gfCNCPoint3[19226] = {X 296.3838, Y 61.4413, Z -4.6667, A 0.000, B 0.000, C 0.000 }
gfCNCPoint3[19227] = {X 295.8066, Y 62.1158, Z -4.6667, A 0.000, B 0.000, C 0.000 }
gfCNCPoint3[19228] = {X 295.1062, Y 62.6612, Z -4.6667, A 0.000, B 0.000, C 0.000 }
gfCNCPoint3[19229] = {X 294.3109, Y 63.0556, Z -4.6667, A 0.000, B 0.000, C 0.000 }
gfCNCPoint3[19230] = {X 293.4528, Y 63.2829, Z -4.6667, A 0.000, B 0.000, C 0.000 }
gfCNCPoint3[19231] = {X 293.4528, Y 92.7108, Z -4.6667, A 0.000, B 0.000, C 0.000 }
gfCNCPoint3[19232] = {X 294.3107, Y 92.9407, Z -4.6667, A 0.000, B 0.000, C 0.000 }
gfCNCPoint3[19233] = {X 295.1055, Y 93.3369, Z -4.6667, A 0.000, B 0.000, C 0.000 }
gfCNCPoint3[19234] = {X 295.8055, Y 93.8837, Z -4.6667, A 0.000, B 0.000, C 0.000 }
gfCNCPoint3[19235] = {X 296.3823, Y 94.5590, Z -4.6667, A 0.000, B 0.000, C 0.000 }
gfCNCPoint3[19236] = {X 296.8130, Y 95.3358, Z -4.6667, A 0.000, B 0.000, C 0.000 }
gfCNCPoint3[19237] = {X 297.0801, Y 96.1828, Z -4.6667, A 0.000, B 0.000, C 0.000 }
gfCNCPoint3[19238] = {X 297.1731, Y 97.0661, Z -4.6667, A 0.000, B 0.000, C 0.000 }
gfCNCPoint3[19239] = {X 297.1731, Y 97.6950, Z -4.6667, A 0.000, B 0.000, C 0.000 }
gfCNCPoint3[19240] = {X 297.6531, Y 97.6950, Z -4.6667, A 0.000, B 0.000, C 0.000 }
gfCNCPoint3[19241] = {X 314.2152, Y 97.6950, Z -4.6667, A 0.000, B 0.000, C 0.000 }
gfCNCPoint3[19242] = {X 313.0166, Y 96.8446, Z -4.6667, A 0.000, B 0.000, C 0.000 }
gfCNCPoint3[19243] = {X 311.8818, Y 95.9106, Z -4.6667, A 0.000, B 0.000, C 0.000 }
gfCNCPoint3[19244] = {X 310.9060, Y 94.9487, Z -4.6667, A 0.000, B 0.000, C 0.000 }
gfCNCPoint3[19245] = {X 310.0416, Y 93.8855, Z -4.6667, A 0.000, B 0.000, C 0.000 }
gfCNCPoint3[19246] = {X 309.2076, Y 92.5708, Z -4.6667, A 0.000, B 0.000, C 0.000 }
gfCNCPoint3[19247] = {X 308.5438, Y 91.1625, Z -4.6667, A 0.000, B 0.000, C 0.000 }
gfCNCPoint3[19248] = {X 308.0605, Y 89.6826, Z -4.6667, A 0.000, B 0.000, C 0.000 }
gfCNCPoint3[19249] = {X 307.7070, Y 88.0127, Z -4.6667, A 0.000, B 0.000, C 0.000 }
gfCNCPoint3[19250] = {X 307.4982, Y 86.3187, Z -4.6667, A 0.000, B 0.000, C 0.000 }
gfCNCPoint3[19251] = {X 307.4354, Y 84.6131, Z -4.6667, A 0.000, B 0.000, C 0.000 }
gfCNCPoint3[19252] = {X 307.4366, Y 63.6743, Z -4.6667, A 0.000, B 0.000, C 0.000 }
gfCNCPoint3[19253] = {X 306.4282, Y 63.3060, Z -4.6667, A 0.000, B 0.000, C 0.000 }
gfCNCPoint3[19254] = {X 305.5247, Y 62.7262, Z -4.6667, A 0.000, B 0.000, C 0.000 }
gfCNCPoint3[19255] = {X 304.7699, Y 61.9628, Z -4.6667, A 0.000, B 0.000, C 0.000 }
gfCNCPoint3[19256] = {X 304.2002, Y 61.0529, Z -4.6667, A 0.000, B 0.000, C 0.000 }
gfCNCPoint3[19257] = {X 303.8433, Y 60.0404, Z -4.6667, A 0.000, B 0.000, C 0.000 }
gfCNCPoint3[19258] = {X 303.7164, Y 58.9744, Z -4.6667, A 0.000, B 0.000, C 0.000 }
gfCNCPoint3[19259] = {X 303.7162, Y 58.0000, Z -4.6667, A 0.000, B 0.000, C 0.000 }
gfCNCPoint3[19260] = {X 303.8100, Y 57.0480, Z -4.6667, A 0.000, B 0.000, C 0.000 }
gfCNCPoint3[19261] = {X 304.0877, Y 56.1325, Z -4.6667, A 0.000, B 0.000, C 0.000 }
gfCNCPoint3[19262] = {X 304.5387, Y 55.2888, Z -4.6667, A 0.000, B 0.000, C 0.000 }
gfCNCPoint3[19263] = {X 305.1455, Y 54.5493, Z -4.6667, A 0.000, B 0.000, C 0.000 }
gfCNCPoint3[19264] = {X 305.8850, Y 53.9424, Z -4.6667, A 0.000, B 0.000, C 0.000 }
gfCNCPoint3[19265] = {X 306.7287, Y 53.4915, Z -4.6667, A 0.000, B 0.000, C 0.000 }
gfCNCPoint3[19266] = {X 307.6442, Y 53.2138, Z -4.6667, A 0.000, B 0.000, C 0.000 }
gfCNCPoint3[19267] = {X 308.5962, Y 53.1200, Z -4.6667, A 0.000, B 0.000, C 0.000 }
gfCNCPoint3[19268] = {X 324.3107, Y 53.1200, Z -4.6667, A 0.000, B 0.000, C 0.000 }
gfCNCPoint3[19269] = {X 325.2627, Y 53.2138, Z -4.6667, A 0.000, B 0.000, C 0.000 }
gfCNCPoint3[19270] = {X 326.1782, Y 53.4915, Z -4.6667, A 0.000, B 0.000, C 0.000 }
gfCNCPoint3[19271] = {X 327.0219, Y 53.9424, Z -4.6667, A 0.000, B 0.000, C 0.000 }
gfCNCPoint3[19272] = {X 327.7614, Y 54.5493, Z -4.6667, A 0.000, B 0.000, C 0.000 }
gfCNCPoint3[19273] = {X 328.3683, Y 55.2888, Z -4.6667, A 0.000, B 0.000, C 0.000 }
gfCNCPoint3[19274] = {X 328.8192, Y 56.1325, Z -4.6667, A 0.000, B 0.000, C 0.000 }
gfCNCPoint3[19275] = {X 329.0969, Y 57.0480, Z -4.6667, A 0.000, B 0.000, C 0.000 }
gfCNCPoint3[19276] = {X 329.1907, Y 58.0000, Z -4.6667, A 0.000, B 0.000, C 0.000 }
gfCNCPoint3[19277] = {X 329.1907, Y 58.9341, Z -4.6667, A 0.000, B 0.000, C 0.000 }
gfCNCPoint3[19278] = {X 329.0671, Y 60.0067, Z -4.6667, A 0.000, B 0.000, C 0.000 }
gfCNCPoint3[19279] = {X 328.7125, Y 61.0265, Z -4.6667, A 0.000, B 0.000, C 0.000 }
gfCNCPoint3[19280] = {X 328.1440, Y 61.9444, Z -4.6667, A 0.000, B 0.000, C 0.000 }
gfCNCPoint3[19281] = {X 327.3888, Y 62.7161, Z -4.6667, A 0.000, B 0.000, C 0.000 }
gfCNCPoint3[19282] = {X 326.4835, Y 63.3044, Z -4.6667, A 0.000, B 0.000, C 0.000 }
gfCNCPoint3[19283] = {X 325.4716, Y 63.6810, Z -4.6667, A 0.000, B 0.000, C 0.000 }
gfCNCPoint3[19284] = {X 325.4732, Y 83.2268, Z -4.6667, A 0.000, B 0.000, C 0.000 }
gfCNCPoint3[19285] = {X 325.4867, Y 84.6073, Z -4.6667, A 0.000, B 0.000, C 0.000 }
gfCNCPoint3[19286] = {X 325.5527, Y 85.7200, Z -4.6667, A 0.000, B 0.000, C 0.000 }
gfCNCPoint3[19287] = {X 325.7426, Y 86.8184, Z -4.6667, A 0.000, B 0.000, C 0.000 }
gfCNCPoint3[19288] = {X 325.8866, Y 86.9525, Z -4.6667, A 0.000, B 0.000, C 0.000 }
gfCNCPoint3[19289] = {X 326.0549, Y 87.0546, Z -4.6667, A 0.000, B 0.000, C 0.000 }
gfCNCPoint3[19290] = {X 326.4838, Y 87.2970, Z -4.6667, A 0.000, B 0.000, C 0.000 }
gfCNCPoint3[19291] = {X 327.8570, Y 87.8652, Z -4.6667, A 0.000, B 0.000, C 0.000 }
gfCNCPoint3[19292] = {X 329.2839, Y 88.2806, Z -4.6667, A 0.000, B 0.000, C 0.000 }
gfCNCPoint3[19293] = {X 332.3217, Y 88.8890, Z -4.6667, A 0.000, B 0.000, C 0.000 }
gfCNCPoint3[19294] = {X 335.3954, Y 89.2771, Z -4.6667, A 0.000, B 0.000, C 0.000 }
gfCNCPoint3[19295] = {X 339.5150, Y 89.5958, Z -4.6667, A 0.000, B 0.000, C 0.000 }
gfCNCPoint3[19296] = {X 343.6430, Y 89.7746, Z -4.6667, A 0.000, B 0.000, C 0.000 }
gfCNCPoint3[19297] = {X 347.7747, Y 89.8134, Z -4.6667, A 0.000, B 0.000, C 0.000 }
gfCNCPoint3[19298] = {X 352.1399, Y 89.7754, Z -4.6667, A 0.000, B 0.000, C 0.000 }
gfCNCPoint3[19299] = {X 356.5008, Y 89.5805, Z -4.6667, A 0.000, B 0.000, C 0.000 }
gfCNCPoint3[19300] = {X 360.8519, Y 89.2288, Z -4.6667, A 0.000, B 0.000, C 0.000 }
gfCNCPoint3[19301] = {X 363.1336, Y 88.9451, Z -4.6667, A 0.000, B 0.000, C 0.000 }
gfCNCPoint3[19302] = {X 365.3941, Y 88.5248, Z -4.6667, A 0.000, B 0.000, C 0.000 }
gfCNCPoint3[19303] = {X 367.6252, Y 87.9694, Z -4.6667, A 0.000, B 0.000, C 0.000 }
gfCNCPoint3[19304] = {X 368.9185, Y 87.4946, Z -4.6667, A 0.000, B 0.000, C 0.000 }
gfCNCPoint3[19305] = {X 370.1140, Y 86.8097, Z -4.6667, A 0.000, B 0.000, C 0.000 }
gfCNCPoint3[19306] = {X 370.2985, Y 85.3241, Z -4.6667, A 0.000, B 0.000, C 0.000 }
gfCNCPoint3[19307] = {X 370.3601, Y 83.8283, Z -4.6667, A 0.000, B 0.000, C 0.000 }
gfCNCPoint3[19308] = {X 370.3587, Y 63.6740, Z -4.6667, A 0.000, B 0.000, C 0.000 }
gfCNCPoint3[19309] = {X 369.3505, Y 63.3056, Z -4.6667, A 0.000, B 0.000, C 0.000 }
gfCNCPoint3[19310] = {X 368.4472, Y 62.7258, Z -4.6667, A 0.000, B 0.000, C 0.000 }
gfCNCPoint3[19311] = {X 367.6926, Y 61.9624, Z -4.6667, A 0.000, B 0.000, C 0.000 }
gfCNCPoint3[19312] = {X 367.1231, Y 61.0526, Z -4.6667, A 0.000, B 0.000, C 0.000 }
gfCNCPoint3[19313] = {X 366.7663, Y 60.0402, Z -4.6667, A 0.000, B 0.000, C 0.000 }
gfCNCPoint3[19314] = {X 366.6394, Y 58.9744, Z -4.6667, A 0.000, B 0.000, C 0.000 }
gfCNCPoint3[19315] = {X 366.6393, Y 58.0000, Z -4.6667, A 0.000, B 0.000, C 0.000 }
gfCNCPoint3[19316] = {X 366.7331, Y 57.0480, Z -4.6667, A 0.000, B 0.000, C 0.000 }
gfCNCPoint3[19317] = {X 367.0108, Y 56.1325, Z -4.6667, A 0.000, B 0.000, C 0.000 }
gfCNCPoint3[19318] = {X 367.4617, Y 55.2888, Z -4.6667, A 0.000, B 0.000, C 0.000 }
gfCNCPoint3[19319] = {X 368.0686, Y 54.5493, Z -4.6667, A 0.000, B 0.000, C 0.000 }
gfCNCPoint3[19320] = {X 368.8081, Y 53.9424, Z -4.6667, A 0.000, B 0.000, C 0.000 }
gfCNCPoint3[19321] = {X 369.6518, Y 53.4915, Z -4.6667, A 0.000, B 0.000, C 0.000 }
gfCNCPoint3[19322] = {X 370.5672, Y 53.2138, Z -4.6667, A 0.000, B 0.000, C 0.000 }
gfCNCPoint3[19323] = {X 371.5193, Y 53.1200, Z -4.6667, A 0.000, B 0.000, C 0.000 }
gfCNCPoint3[19324] = {X 388.0597, Y 53.1200, Z -4.6667, A 0.000, B 0.000, C 0.000 }
gfCNCPoint3[19325] = {X 389.0355, Y 53.2186, Z -4.6667, A 0.000, B 0.000, C 0.000 }
gfCNCPoint3[19326] = {X 389.9719, Y 53.5102, Z -4.6667, A 0.000, B 0.000, C 0.000 }
gfCNCPoint3[19327] = {X 390.8310, Y 53.9833, Z -4.6667, A 0.000, B 0.000, C 0.000 }
gfCNCPoint3[19328] = {X 391.5783, Y 54.6186, Z -4.6667, A 0.000, B 0.000, C 0.000 }
gfCNCPoint3[19329] = {X 392.1572, Y 55.3496, Z -4.6667, A 0.000, B 0.000, C 0.000 }
gfCNCPoint3[19330] = {X 392.5865, Y 56.1774, Z -4.6667, A 0.000, B 0.000, C 0.000 }
gfCNCPoint3[19331] = {X 392.8506, Y 57.0718, Z -4.6667, A 0.000, B 0.000, C 0.000 }
gfCNCPoint3[19332] = {X 392.9397, Y 58.0000, Z -4.6667, A 0.000, B 0.000, C 0.000 }
gfCNCPoint3[19333] = {X 392.9395, Y 58.9743, Z -4.6667, A 0.000, B 0.000, C 0.000 }
gfCNCPoint3[19334] = {X 392.8783, Y 59.7057, Z -4.6667, A 0.000, B 0.000, C 0.000 }
gfCNCPoint3[19335] = {X 392.7080, Y 60.4197, Z -4.6667, A 0.000, B 0.000, C 0.000 }
gfCNCPoint3[19336] = {X 392.4327, Y 61.1000, Z -4.6667, A 0.000, B 0.000, C 0.000 }
gfCNCPoint3[19337] = {X 392.0515, Y 61.7416, Z -4.6667, A 0.000, B 0.000, C 0.000 }
gfCNCPoint3[19338] = {X 391.5775, Y 62.3178, Z -4.6667, A 0.000, B 0.000, C 0.000 }
gfCNCPoint3[19339] = {X 390.8819, Y 62.9185, Z -4.6667, A 0.000, B 0.000, C 0.000 }
gfCNCPoint3[19340] = {X 390.0864, Y 63.3788, Z -4.6667, A 0.000, B 0.000, C 0.000 }
gfCNCPoint3[19341] = {X 389.2190, Y 63.6825, Z -4.6667, A 0.000, B 0.000, C 0.000 }
gfCNCPoint3[19342] = {X 389.2180, Y 73.4816, Z -4.6667, A 0.000, B 0.000, C 0.000 }
gfCNCPoint3[19343] = {X 398.8180, Y 73.4825, Z -4.6667, A 0.000, B 0.000, C 0.000 }
gfCNCPoint3[19344] = {X 398.8173, Y 80.5578, Z -4.6667, A 0.000, B 0.000, C 0.000 }
gfCNCPoint3[19345] = {X 405.8037, Y 76.0835, Z -4.6667, A 0.000, B 0.000, C 0.000 }
gfCNCPoint3[19346] = {X 400.0374, Y 73.8211, Z -4.6667, A 0.000, B 0.000, C 0.000 }
gfCNCPoint3[19347] = {X 399.4365, Y 73.6201, Z -4.6667, A 0.000, B 0.000, C 0.000 }
gfCNCPoint3[19348] = {X 398.8180, Y 73.4825, Z -4.6667, A 0.000, B 0.000, C 0.000 }
gfCNCPoint3[19349] = {X 396.4180, Y 73.4822, Z -4.6667, A 0.000, B 0.000, C 0.000 }
gfCNCPoint3[19350] = {X 396.4170, Y 84.5897, Z -4.6667, A 0.000, B 0.000, C 0.000 }
gfCNCPoint3[19351] = {X 396.4168, Y 84.9452, Z -4.6667, A 0.000, B 0.000, C 0.000 }
gfCNCPoint3[19352] = {X 411.0595, Y 75.5675, Z -4.6667, A 0.000, B 0.000, C 0.000 }
gfCNCPoint3[19353] = {X 400.9158, Y 71.5876, Z -4.6667, A 0.000, B 0.000, C 0.000 }
gfCNCPoint3[19354] = {X 399.6202, Y 71.1939, Z -4.6667, A 0.000, B 0.000, C 0.000 }
gfCNCPoint3[19355] = {X 398.2786, Y 71.0108, Z -4.6667, A 0.000, B 0.000, C 0.000 }
gfCNCPoint3[19356] = {X 397.3448, Y 70.9530, Z -4.6667, A 0.000, B 0.000, C 0.000 }
gfCNCPoint3[19357] = {X 396.4183, Y 70.8231, Z -4.6667, A 0.000, B 0.000, C 0.000 }
gfCNCPoint3[19358] = {X 396.4180, Y 73.4822, Z -4.6667, A 0.000, B 0.000, C 0.000 }
gfCNCPoint3[19359] = {X 394.0180, Y 73.4820, Z -4.6667, A 0.000, B 0.000, C 0.000 }
gfCNCPoint3[19360] = {X 394.0170, Y 84.5974, Z -4.6667, A 0.000, B 0.000, C 0.000 }
gfCNCPoint3[19361] = {X 394.0175, Y 84.7629, Z -4.6667, A 0.000, B 0.000, C 0.000 }
gfCNCPoint3[19362] = {X 394.0169, Y 84.9284, Z -4.6667, A 0.000, B 0.000, C 0.000 }
gfCNCPoint3[19363] = {X 393.9665, Y 86.3336, Z -4.6667, A 0.000, B 0.000, C 0.000 }
gfCNCPoint3[19364] = {X 393.8352, Y 87.7335, Z -4.6667, A 0.000, B 0.000, C 0.000 }
gfCNCPoint3[19365] = {X 395.0900, Y 87.4758, Z -4.6667, A 0.000, B 0.000, C 0.000 }
gfCNCPoint3[19366] = {X 396.3680, Y 87.3860, Z -4.6667, A 0.000, B 0.000, C 0.000 }
gfCNCPoint3[19367] = {X 396.7432, Y 87.3712, Z -4.6667, A 0.000, B 0.000, C 0.000 }
gfCNCPoint3[19368] = {X 397.1178, Y 87.3462, Z -4.6667, A 0.000, B 0.000, C 0.000 }
gfCNCPoint3[19369] = {X 416.3153, Y 75.0514, Z -4.6667, A 0.000, B 0.000, C 0.000 }
gfCNCPoint3[19370] = {X 401.7941, Y 69.3541, Z -4.6667, A 0.000, B 0.000, C 0.000 }
gfCNCPoint3[19371] = {X 400.6812, Y 68.9842, Z -4.6667, A 0.000, B 0.000, C 0.000 }
gfCNCPoint3[19372] = {X 399.5351, Y 68.7359, Z -4.6667, A 0.000, B 0.000, C 0.000 }
gfCNCPoint3[19373] = {X 398.3689, Y 68.6122, Z -4.6667, A 0.000, B 0.000, C 0.000 }
gfCNCPoint3[19374] = {X 397.6031, Y 68.5669, Z -4.6667, A 0.000, B 0.000, C 0.000 }
gfCNCPoint3[19375] = {X 396.8433, Y 68.4610, Z -4.6667, A 0.000, B 0.000, C 0.000 }
gfCNCPoint3[19376] = {X 395.3930, Y 68.0821, Z -4.6667, A 0.000, B 0.000, C 0.000 }
gfCNCPoint3[19377] = {X 394.0186, Y 67.4838, Z -4.6667, A 0.000, B 0.000, C 0.000 }
gfCNCPoint3[19378] = {X 394.0180, Y 73.4820, Z -4.6667, A 0.000, B 0.000, C 0.000 }
gfCNCPoint3[19379] = {X 391.6180, Y 73.4818, Z -4.6667, A 0.000, B 0.000, C 0.000 }
gfCNCPoint3[19380] = {X 391.6169, Y 84.6054, Z -4.6667, A 0.000, B 0.000, C 0.000 }
gfCNCPoint3[19381] = {X 391.5809, Y 86.0256, Z -4.6667, A 0.000, B 0.000, C 0.000 }
gfCNCPoint3[19382] = {X 391.4531, Y 87.4405, Z -4.6667, A 0.000, B 0.000, C 0.000 }
gfCNCPoint3[19383] = {X 391.2288, Y 88.8722, Z -4.6667, A 0.000, B 0.000, C 0.000 }
gfCNCPoint3[19384] = {X 390.9106, Y 90.2860, Z -4.6667, A 0.000, B 0.000, C 0.000 }
gfCNCPoint3[19385] = {X 390.3344, Y 92.0499, Z -4.6667, A 0.000, B 0.000, C 0.000 }
gfCNCPoint3[19386] = {X 389.5429, Y 93.7283, Z -4.6667, A 0.000, B 0.000, C 0.000 }
gfCNCPoint3[19387] = {X 388.5486, Y 95.2950, Z -4.6667, A 0.000, B 0.000, C 0.000 }
gfCNCPoint3[19388] = {X 389.3446, Y 95.2950, Z -4.6667, A 0.000, B 0.000, C 0.000 }
gfCNCPoint3[19389] = {X 389.7639, Y 94.0857, Z -4.6667, A 0.000, B 0.000, C 0.000 }
gfCNCPoint3[19390] = {X 390.3885, Y 92.9685, Z -4.6667, A 0.000, B 0.000, C 0.000 }
gfCNCPoint3[19391] = {X 391.1991, Y 91.9779, Z -4.6667, A 0.000, B 0.000, C 0.000 }
gfCNCPoint3[19392] = {X 392.1707, Y 91.1447, Z -4.6667, A 0.000, B 0.000, C 0.000 }
gfCNCPoint3[19393] = {X 393.2732, Y 90.4945, Z -4.6667, A 0.000, B 0.000, C 0.000 }
gfCNCPoint3[19394] = {X 394.4725, Y 90.0474, Z -4.6667, A 0.000, B 0.000, C 0.000 }
gfCNCPoint3[19395] = {X 395.4279, Y 89.8519, Z -4.6667, A 0.000, B 0.000, C 0.000 }
gfCNCPoint3[19396] = {X 396.4007, Y 89.7859, Z -4.6667, A 0.000, B 0.000, C 0.000 }
gfCNCPoint3[19397] = {X 397.1636, Y 89.7496, Z -4.6667, A 0.000, B 0.000, C 0.000 }
gfCNCPoint3[19398] = {X 397.9239, Y 89.6774, Z -4.6667, A 0.000, B 0.000, C 0.000 }
gfCNCPoint3[19399] = {X 417.6096, Y 77.0725, Z -4.6667, A 0.000, B 0.000, C 0.000 }
gfCNCPoint3[19400] = {X 421.5711, Y 74.5354, Z -4.6667, A 0.000, B 0.000, C 0.000 }
gfCNCPoint3[19401] = {X 402.6725, Y 67.1206, Z -4.6667, A 0.000, B 0.000, C 0.000 }
gfCNCPoint3[19402] = {X 401.3007, Y 66.6655, Z -4.6667, A 0.000, B 0.000, C 0.000 }
gfCNCPoint3[19403] = {X 399.8876, Y 66.3618, Z -4.6667, A 0.000, B 0.000, C 0.000 }
gfCNCPoint3[19404] = {X 398.4499, Y 66.2133, Z -4.6667, A 0.000, B 0.000, C 0.000 }
gfCNCPoint3[19405] = {X 397.3054, Y 66.1055, Z -4.6667, A 0.000, B 0.000, C 0.000 }
gfCNCPoint3[19406] = {X 396.1922, Y 65.8190, Z -4.6667, A 0.000, B 0.000, C 0.000 }
gfCNCPoint3[19407] = {X 395.1380, Y 65.3609, Z -4.6667, A 0.000, B 0.000, C 0.000 }
gfCNCPoint3[19408] = {X 394.1690, Y 64.7424, Z -4.6667, A 0.000, B 0.000, C 0.000 }
gfCNCPoint3[19409] = {X 393.3094, Y 63.9792, Z -4.6667, A 0.000, B 0.000, C 0.000 }
gfCNCPoint3[19410] = {X 392.5123, Y 64.6964, Z -4.6667, A 0.000, B 0.000, C 0.000 }
gfCNCPoint3[19411] = {X 391.6188, Y 65.2892, Z -4.6667, A 0.000, B 0.000, C 0.000 }
gfCNCPoint3[19412] = {X 391.6180, Y 73.4818, Z -4.6667, A 0.000, B 0.000, C 0.000 }
gfCNCPoint3[19413] = {X 389.2180, Y 73.4816, Z -4.6667, A 0.000, B 0.000, C 0.000 }
gfCNCPoint3[19414] = {X 389.2169, Y 84.6139, Z -4.6667, A 0.000, B 0.000, C 0.000 }
gfCNCPoint3[19415] = {X 389.1551, Y 86.3199, Z -4.6667, A 0.000, B 0.000, C 0.000 }
gfCNCPoint3[19416] = {X 388.9447, Y 88.0140, Z -4.6667, A 0.000, B 0.000, C 0.000 }
gfCNCPoint3[19417] = {X 388.5875, Y 89.6833, Z -4.6667, A 0.000, B 0.000, C 0.000 }
gfCNCPoint3[19418] = {X 388.1043, Y 91.1629, Z -4.6667, A 0.000, B 0.000, C 0.000 }
gfCNCPoint3[19419] = {X 387.4405, Y 92.5708, Z -4.6667, A 0.000, B 0.000, C 0.000 }
gfCNCPoint3[19420] = {X 386.6065, Y 93.8850, Z -4.6667, A 0.000, B 0.000, C 0.000 }
gfCNCPoint3[19421] = {X 385.8743, Y 94.7997, Z -4.6667, A 0.000, B 0.000, C 0.000 }
gfCNCPoint3[19422] = {X 385.0595, Y 95.6417, Z -4.6667, A 0.000, B 0.000, C 0.000 }
gfCNCPoint3[19423] = {X 383.7996, Y 96.7249, Z -4.6667, A 0.000, B 0.000, C 0.000 }
gfCNCPoint3[19424] = {X 382.4506, Y 97.6950, Z -4.6667, A 0.000, B 0.000, C 0.000 }
gfCNCPoint3[19425] = {X 382.1875, Y 97.2936, Z -4.6667, A 0.000, B 0.000, C 0.000 }
gfCNCPoint3[19426] = {X 381.0199, Y 97.9993, Z -4.6667, A 0.000, B 0.000, C 0.000 }
gfCNCPoint3[19427] = {X 379.8040, Y 98.6181, Z -4.6667, A 0.000, B 0.000, C 0.000 }
gfCNCPoint3[19428] = {X 377.5271, Y 99.5766, Z -4.6667, A 0.000, B 0.000, C 0.000 }
gfCNCPoint3[19429] = {X 375.1871, Y 100.3689, Z -4.6667, A 0.000, B 0.000, C 0.000 }
gfCNCPoint3[19430] = {X 372.7962, Y 100.9907, Z -4.6667, A 0.000, B 0.000, C 0.000 }
gfCNCPoint3[19431] = {X 368.8820, Y 101.7454, Z -4.6667, A 0.000, B 0.000, C 0.000 }
gfCNCPoint3[19432] = {X 364.9353, Y 102.3062, Z -4.6667, A 0.000, B 0.000, C 0.000 }
gfCNCPoint3[19433] = {X 360.9658, Y 102.6716, Z -4.6667, A 0.000, B 0.000, C 0.000 }
gfCNCPoint3[19434] = {X 355.2455, Y 102.9767, Z -4.6667, A 0.000, B 0.000, C 0.000 }
gfCNCPoint3[19435] = {X 349.5185, Y 103.1068, Z -4.6667, A 0.000, B 0.000, C 0.000 }
gfCNCPoint3[19436] = {X 343.7903, Y 103.0618, Z -4.6667, A 0.000, B 0.000, C 0.000 }
gfCNCPoint3[19437] = {X 338.0661, Y 102.8417, Z -4.6667, A 0.000, B 0.000, C 0.000 }
gfCNCPoint3[19438] = {X 334.1085, Y 102.5645, Z -4.6667, A 0.000, B 0.000, C 0.000 }
gfCNCPoint3[19439] = {X 330.1660, Y 102.1223, Z -4.6667, A 0.000, B 0.000, C 0.000 }
gfCNCPoint3[19440] = {X 326.2454, Y 101.5158, Z -4.6667, A 0.000, B 0.000, C 0.000 }
gfCNCPoint3[19441] = {X 323.3898, Y 100.9107, Z -4.6667, A 0.000, B 0.000, C 0.000 }
gfCNCPoint3[19442] = {X 320.5867, Y 100.0961, Z -4.6667, A 0.000, B 0.000, C 0.000 }
gfCNCPoint3[19443] = {X 317.8516, Y 99.0765, Z -4.6667, A 0.000, B 0.000, C 0.000 }
gfCNCPoint3[19444] = {X 316.3332, Y 98.3751, Z -4.6667, A 0.000, B 0.000, C 0.000 }
gfCNCPoint3[19445] = {X 314.8785, Y 97.5498, Z -4.6667, A 0.000, B 0.000, C 0.000 }
gfCNCPoint3[19446] = {X 313.4975, Y 96.6063, Z -4.6667, A 0.000, B 0.000, C 0.000 }
gfCNCPoint3[19447] = {X 312.1998, Y 95.5512, Z -4.6667, A 0.000, B 0.000, C 0.000 }
gfCNCPoint3[19448] = {X 311.1892, Y 94.5459, Z -4.6667, A 0.000, B 0.000, C 0.000 }
gfCNCPoint3[19449] = {X 310.3050, Y 93.4278, Z -4.6667, A 0.000, B 0.000, C 0.000 }
gfCNCPoint3[19450] = {X 309.5595, Y 92.2128, Z -4.6667, A 0.000, B 0.000, C 0.000 }
gfCNCPoint3[19451] = {X 308.9634, Y 90.9180, Z -4.6667, A 0.000, B 0.000, C 0.000 }
gfCNCPoint3[19452] = {X 308.5250, Y 89.5616, Z -4.6667, A 0.000, B 0.000, C 0.000 }
gfCNCPoint3[19453] = {X 308.1802, Y 87.9321, Z -4.6667, A 0.000, B 0.000, C 0.000 }
gfCNCPoint3[19454] = {X 307.9765, Y 86.2791, Z -4.6667, A 0.000, B 0.000, C 0.000 }
gfCNCPoint3[19455] = {X 307.9154, Y 84.6146, Z -4.6667, A 0.000, B 0.000, C 0.000 }
gfCNCPoint3[19456] = {X 307.9166, Y 63.2813, Z -4.6667, A 0.000, B 0.000, C 0.000 }
gfCNCPoint3[19457] = {X 307.0573, Y 63.0561, Z -4.6667, A 0.000, B 0.000, C 0.000 }
gfCNCPoint3[19458] = {X 306.2606, Y 62.6630, Z -4.6667, A 0.000, B 0.000, C 0.000 }
gfCNCPoint3[19459] = {X 305.5592, Y 62.1178, Z -4.6667, A 0.000, B 0.000, C 0.000 }
gfCNCPoint3[19460] = {X 304.9816, Y 61.4429, Z -4.6667, A 0.000, B 0.000, C 0.000 }
gfCNCPoint3[19461] = {X 304.5513, Y 60.6657, Z -4.6667, A 0.000, B 0.000, C 0.000 }
gfCNCPoint3[19462] = {X 304.2859, Y 59.8179, Z -4.6667, A 0.000, B 0.000, C 0.000 }
gfCNCPoint3[19463] = {X 304.1962, Y 58.9341, Z -4.6667, A 0.000, B 0.000, C 0.000 }
gfCNCPoint3[19464] = {X 304.1962, Y 58.0000, Z -4.6667, A 0.000, B 0.000, C 0.000 }
gfCNCPoint3[19465] = {X 304.3065, Y 57.0209, Z -4.6667, A 0.000, B 0.000, C 0.000 }
gfCNCPoint3[19466] = {X 304.6320, Y 56.0909, Z -4.6667, A 0.000, B 0.000, C 0.000 }
gfCNCPoint3[19467] = {X 305.1562, Y 55.2566, Z -4.6667, A 0.000, B 0.000, C 0.000 }
gfCNCPoint3[19468] = {X 305.8529, Y 54.5599, Z -4.6667, A 0.000, B 0.000, C 0.000 }
gfCNCPoint3[19469] = {X 306.6871, Y 54.0357, Z -4.6667, A 0.000, B 0.000, C 0.000 }
gfCNCPoint3[19470] = {X 307.6171, Y 53.7103, Z -4.6667, A 0.000, B 0.000, C 0.000 }
gfCNCPoint3[19471] = {X 308.5962, Y 53.6000, Z -4.6667, A 0.000, B 0.000, C 0.000 }
gfCNCPoint3[19472] = {X 324.3107, Y 53.6000, Z -4.6667, A 0.000, B 0.000, C 0.000 }
gfCNCPoint3[19473] = {X 325.2898, Y 53.7103, Z -4.6667, A 0.000, B 0.000, C 0.000 }
gfCNCPoint3[19474] = {X 326.2198, Y 54.0357, Z -4.6667, A 0.000, B 0.000, C 0.000 }
gfCNCPoint3[19475] = {X 327.0540, Y 54.5599, Z -4.6667, A 0.000, B 0.000, C 0.000 }
gfCNCPoint3[19476] = {X 327.7507, Y 55.2566, Z -4.6667, A 0.000, B 0.000, C 0.000 }
gfCNCPoint3[19477] = {X 328.2750, Y 56.0909, Z -4.6667, A 0.000, B 0.000, C 0.000 }
gfCNCPoint3[19478] = {X 328.6004, Y 57.0209, Z -4.6667, A 0.000, B 0.000, C 0.000 }
gfCNCPoint3[19479] = {X 328.7107, Y 58.0000, Z -4.6667, A 0.000, B 0.000, C 0.000 }
gfCNCPoint3[19480] = {X 328.7107, Y 58.9364, Z -4.6667, A 0.000, B 0.000, C 0.000 }
gfCNCPoint3[19481] = {X 328.6169, Y 59.8191, Z -4.6667, A 0.000, B 0.000, C 0.000 }
gfCNCPoint3[19482] = {X 328.3493, Y 60.6655, Z -4.6667, A 0.000, B 0.000, C 0.000 }
gfCNCPoint3[19483] = {X 327.9186, Y 61.4417, Z -4.6667, A 0.000, B 0.000, C 0.000 }
gfCNCPoint3[19484] = {X 327.3421, Y 62.1166, Z -4.6667, A 0.000, B 0.000, C 0.000 }
gfCNCPoint3[19485] = {X 326.6428, Y 62.6634, Z -4.6667, A 0.000, B 0.000, C 0.000 }
gfCNCPoint3[19486] = {X 325.8487, Y 63.0601, Z -4.6667, A 0.000, B 0.000, C 0.000 }
gfCNCPoint3[19487] = {X 324.9916, Y 63.2908, Z -4.6667, A 0.000, B 0.000, C 0.000 }
gfCNCPoint3[19488] = {X 324.9932, Y 83.2292, Z -4.6667, A 0.000, B 0.000, C 0.000 }
gfCNCPoint3[19489] = {X 325.0068, Y 84.6144, Z -4.6667, A 0.000, B 0.000, C 0.000 }
gfCNCPoint3[19490] = {X 325.0826, Y 85.8324, Z -4.6667, A 0.000, B 0.000, C 0.000 }
gfCNCPoint3[19491] = {X 325.3002, Y 87.0333, Z -4.6667, A 0.000, B 0.000, C 0.000 }
gfCNCPoint3[19492] = {X 325.5332, Y 87.2838, Z -4.6667, A 0.000, B 0.000, C 0.000 }
gfCNCPoint3[19493] = {X 325.8187, Y 87.4724, Z -4.6667, A 0.000, B 0.000, C 0.000 }
gfCNCPoint3[19494] = {X 326.2616, Y 87.7228, Z -4.6667, A 0.000, B 0.000, C 0.000 }
gfCNCPoint3[19495] = {X 327.6911, Y 88.3157, Z -4.6667, A 0.000, B 0.000, C 0.000 }
gfCNCPoint3[19496] = {X 329.1769, Y 88.7485, Z -4.6667, A 0.000, B 0.000, C 0.000 }
gfCNCPoint3[19497] = {X 332.2475, Y 89.3632, Z -4.6667, A 0.000, B 0.000, C 0.000 }
gfCNCPoint3[19498] = {X 335.3543, Y 89.7554, Z -4.6667, A 0.000, B 0.000, C 0.000 }
gfCNCPoint3[19499] = {X 339.4910, Y 90.0752, Z -4.6667, A 0.000, B 0.000, C 0.000 }
gfCNCPoint3[19500] = {X 343.6362, Y 90.2546, Z -4.6667, A 0.000, B 0.000, C 0.000 }
gfCNCPoint3[19501] = {X 347.7851, Y 90.2934, Z -4.6667, A 0.000, B 0.000, C 0.000 }
gfCNCPoint3[19502] = {X 352.1632, Y 90.2549, Z -4.6667, A 0.000, B 0.000, C 0.000 }
gfCNCPoint3[19503] = {X 356.5371, Y 90.0591, Z -4.6667, A 0.000, B 0.000, C 0.000 }
gfCNCPoint3[19504] = {X 360.9012, Y 89.7062, Z -4.6667, A 0.000, B 0.000, C 0.000 }
gfCNCPoint3[19505] = {X 363.2108, Y 89.4189, Z -4.6667, A 0.000, B 0.000, C 0.000 }
gfCNCPoint3[19506] = {X 365.4989, Y 88.9933, Z -4.6667, A 0.000, B 0.000, C 0.000 }
gfCNCPoint3[19507] = {X 367.7574, Y 88.4308, Z -4.6667, A 0.000, B 0.000, C 0.000 }
gfCNCPoint3[19508] = {X 368.6801, Y 88.1205, Z -4.6667, A 0.000, B 0.000, C 0.000 }
gfCNCPoint3[19509] = {X 369.5623, Y 87.7087, Z -4.6667, A 0.000, B 0.000, C 0.000 }
gfCNCPoint3[19510] = {X 370.3927, Y 87.2006, Z -4.6667, A 0.000, B 0.000, C 0.000 }
gfCNCPoint3[19511] = {X 370.5205, Y 87.0676, Z -4.6667, A 0.000, B 0.000, C 0.000 }
gfCNCPoint3[19512] = {X 370.5863, Y 86.8954, Z -4.6667, A 0.000, B 0.000, C 0.000 }
gfCNCPoint3[19513] = {X 370.7766, Y 85.3671, Z -4.6667, A 0.000, B 0.000, C 0.000 }
gfCNCPoint3[19514] = {X 370.8401, Y 83.8283, Z -4.6667, A 0.000, B 0.000, C 0.000 }
gfCNCPoint3[19515] = {X 370.8386, Y 63.2811, Z -4.6667, A 0.000, B 0.000, C 0.000 }
gfCNCPoint3[19516] = {X 369.9795, Y 63.0558, Z -4.6667, A 0.000, B 0.000, C 0.000 }
gfCNCPoint3[19517] = {X 369.1830, Y 62.6626, Z -4.6667, A 0.000, B 0.000, C 0.000 }
gfCNCPoint3[19518] = {X 368.4818, Y 62.1174, Z -4.6667, A 0.000, B 0.000, C 0.000 }
gfCNCPoint3[19519] = {X 367.9044, Y 61.4425, Z -4.6667, A 0.000, B 0.000, C 0.000 }
gfCNCPoint3[19520] = {X 367.4742, Y 60.6654, Z -4.6667, A 0.000, B 0.000, C 0.000 }
gfCNCPoint3[19521] = {X 367.2089, Y 59.8177, Z -4.6667, A 0.000, B 0.000, C 0.000 }
gfCNCPoint3[19522] = {X 367.1193, Y 58.9340, Z -4.6667, A 0.000, B 0.000, C 0.000 }
gfCNCPoint3[19523] = {X 367.1193, Y 58.0000, Z -4.6667, A 0.000, B 0.000, C 0.000 }
gfCNCPoint3[19524] = {X 367.2296, Y 57.0209, Z -4.6667, A 0.000, B 0.000, C 0.000 }
gfCNCPoint3[19525] = {X 367.5550, Y 56.0909, Z -4.6667, A 0.000, B 0.000, C 0.000 }
gfCNCPoint3[19526] = {X 368.0792, Y 55.2566, Z -4.6667, A 0.000, B 0.000, C 0.000 }
gfCNCPoint3[19527] = {X 368.7759, Y 54.5599, Z -4.6667, A 0.000, B 0.000, C 0.000 }
gfCNCPoint3[19528] = {X 369.6102, Y 54.0357, Z -4.6667, A 0.000, B 0.000, C 0.000 }
gfCNCPoint3[19529] = {X 370.5402, Y 53.7103, Z -4.6667, A 0.000, B 0.000, C 0.000 }
gfCNCPoint3[19530] = {X 371.5193, Y 53.6000, Z -4.6667, A 0.000, B 0.000, C 0.000 }
gfCNCPoint3[19531] = {X 388.0597, Y 53.6000, Z -4.6667, A 0.000, B 0.000, C 0.000 }
gfCNCPoint3[19532] = {X 389.0388, Y 53.7103, Z -4.6667, A 0.000, B 0.000, C 0.000 }
gfCNCPoint3[19533] = {X 389.9688, Y 54.0357, Z -4.6667, A 0.000, B 0.000, C 0.000 }
gfCNCPoint3[19534] = {X 390.8030, Y 54.5599, Z -4.6667, A 0.000, B 0.000, C 0.000 }
gfCNCPoint3[19535] = {X 391.4997, Y 55.2566, Z -4.6667, A 0.000, B 0.000, C 0.000 }
gfCNCPoint3[19536] = {X 392.0239, Y 56.0909, Z -4.6667, A 0.000, B 0.000, C 0.000 }
gfCNCPoint3[19537] = {X 392.3494, Y 57.0209, Z -4.6667, A 0.000, B 0.000, C 0.000 }
gfCNCPoint3[19538] = {X 392.4597, Y 58.0000, Z -4.6667, A 0.000, B 0.000, C 0.000 }
gfCNCPoint3[19539] = {X 392.4595, Y 58.9704, Z -4.6667, A 0.000, B 0.000, C 0.000 }
gfCNCPoint3[19540] = {X 392.3397, Y 59.9546, Z -4.6667, A 0.000, B 0.000, C 0.000 }
gfCNCPoint3[19541] = {X 392.0025, Y 60.8870, Z -4.6667, A 0.000, B 0.000, C 0.000 }
gfCNCPoint3[19542] = {X 391.5594, Y 61.6016, Z -4.6667, A 0.000, B 0.000, C 0.000 }
gfCNCPoint3[19543] = {X 390.9890, Y 62.2194, Z -4.6667, A 0.000, B 0.000, C 0.000 }
gfCNCPoint3[19544] = {X 390.3120, Y 62.7180, Z -4.6667, A 0.000, B 0.000, C 0.000 }
gfCNCPoint3[19545] = {X 389.5528, Y 63.0795, Z -4.6667, A 0.000, B 0.000, C 0.000 }
gfCNCPoint3[19546] = {X 388.7390, Y 63.2908, Z -4.6667, A 0.000, B 0.000, C 0.000 }
gfCNCPoint3[19547] = {X 388.7390, Y 83.9247, Z -4.6667, A 0.000, B 0.000, C 0.000 }
gfCNCPoint3[19548] = {X 388.7369, Y 84.6150, Z -4.6667, A 0.000, B 0.000, C 0.000 }
gfCNCPoint3[19549] = {X 388.6767, Y 86.2799, Z -4.6667, A 0.000, B 0.000, C 0.000 }
gfCNCPoint3[19550] = {X 388.4716, Y 87.9333, Z -4.6667, A 0.000, B 0.000, C 0.000 }
gfCNCPoint3[19551] = {X 388.1230, Y 89.5625, Z -4.6667, A 0.000, B 0.000, C 0.000 }
gfCNCPoint3[19552] = {X 387.5872, Y 91.1606, Z -4.6667, A 0.000, B 0.000, C 0.000 }
gfCNCPoint3[19553] = {X 386.8325, Y 92.6678, Z -4.6667, A 0.000, B 0.000, C 0.000 }
gfCNCPoint3[19554] = {X 385.8739, Y 94.0542, Z -4.6667, A 0.000, B 0.000, C 0.000 }
gfCNCPoint3[19555] = {X 384.7302, Y 95.2924, Z -4.6667, A 0.000, B 0.000, C 0.000 }
gfCNCPoint3[19556] = {X 383.5022, Y 96.3481, Z -4.6667, A 0.000, B 0.000, C 0.000 }
gfCNCPoint3[19557] = {X 382.1875, Y 97.2936, Z -4.6667, A 0.000, B 0.000, C 0.000 }
gfCNCPoint3[19558] = {X 382.4506, Y 97.6950, Z -4.6667, A 0.000, B 0.000, C 0.000 }
gfCNCPoint3[19559] = {X 391.5259, Y 97.6950, Z -4.6667, A 0.000, B 0.000, C 0.000 }
gfCNCPoint3[19560] = {X 391.5259, Y 97.0659, Z -4.6667, A 0.000, B 0.000, C 0.000 }
gfCNCPoint3[19561] = {X 391.6202, Y 96.1114, Z -4.6667, A 0.000, B 0.000, C 0.000 }
gfCNCPoint3[19562] = {X 391.8994, Y 95.1937, Z -4.6667, A 0.000, B 0.000, C 0.000 }
gfCNCPoint3[19563] = {X 392.3527, Y 94.3483, Z -4.6667, A 0.000, B 0.000, C 0.000 }
gfCNCPoint3[19564] = {X 392.9626, Y 93.6079, Z -4.6667, A 0.000, B 0.000, C 0.000 }
gfCNCPoint3[19565] = {X 393.7055, Y 93.0012, Z -4.6667, A 0.000, B 0.000, C 0.000 }
gfCNCPoint3[19566] = {X 394.5528, Y 92.5515, Z -4.6667, A 0.000, B 0.000, C 0.000 }
gfCNCPoint3[19567] = {X 395.4717, Y 92.2762, Z -4.6667, A 0.000, B 0.000, C 0.000 }
gfCNCPoint3[19568] = {X 396.4267, Y 92.1860, Z -4.6667, A 0.000, B 0.000, C 0.000 }
gfCNCPoint3[19569] = {X 397.3274, Y 92.1440, Z -4.6667, A 0.000, B 0.000, C 0.000 }
gfCNCPoint3[19570] = {X 398.2250, Y 92.0585, Z -4.6667, A 0.000, B 0.000, C 0.000 }
gfCNCPoint3[19571] = {X 398.7531, Y 91.9301, Z -4.6667, A 0.000, B 0.000, C 0.000 }
gfCNCPoint3[19572] = {X 399.2394, Y 91.6875, Z -4.6667, A 0.000, B 0.000, C 0.000 }
gfCNCPoint3[19573] = {X 426.8269, Y 74.0194, Z -4.6667, A 0.000, B 0.000, C 0.000 }
gfCNCPoint3[19574] = {X 403.5509, Y 64.8871, Z -4.6667, A 0.000, B 0.000, C 0.000 }
gfCNCPoint3[19575] = {X 401.9167, Y 64.3458, Z -4.6667, A 0.000, B 0.000, C 0.000 }
gfCNCPoint3[19576] = {X 400.2331, Y 63.9867, Z -4.6667, A 0.000, B 0.000, C 0.000 }
gfCNCPoint3[19577] = {X 398.5203, Y 63.8139, Z -4.6667, A 0.000, B 0.000, C 0.000 }
gfCNCPoint3[19578] = {X 397.5546, Y 63.7099, Z -4.6667, A 0.000, B 0.000, C 0.000 }
gfCNCPoint3[19579] = {X 396.6286, Y 63.4166, Z -4.6667, A 0.000, B 0.000, C 0.000 }
gfCNCPoint3[19580] = {X 395.7791, Y 62.9457, Z -4.6667, A 0.000, B 0.000, C 0.000 }
gfCNCPoint3[19581] = {X 395.0396, Y 62.3160, Z -4.6667, A 0.000, B 0.000, C 0.000 }
gfCNCPoint3[19582] = {X 394.4660, Y 61.5934, Z -4.6667, A 0.000, B 0.000, C 0.000 }
gfCNCPoint3[19583] = {X 394.0386, Y 60.7757, Z -4.6667, A 0.000, B 0.000, C 0.000 }
gfCNCPoint3[19584] = {X 393.7727, Y 59.8921, Z -4.6667, A 0.000, B 0.000, C 0.000 }
gfCNCPoint3[19585] = {X 393.6779, Y 58.9744, Z -4.6667, A 0.000, B 0.000, C 0.000 }
gfCNCPoint3[19586] = {X 393.6777, Y 58.0000, Z -4.6667, A 0.000, B 0.000, C 0.000 }
gfCNCPoint3[19587] = {X 393.7668, Y 57.0718, Z -4.6667, A 0.000, B 0.000, C 0.000 }
gfCNCPoint3[19588] = {X 394.0309, Y 56.1774, Z -4.6667, A 0.000, B 0.000, C 0.000 }
gfCNCPoint3[19589] = {X 394.4602, Y 55.3496, Z -4.6667, A 0.000, B 0.000, C 0.000 }
gfCNCPoint3[19590] = {X 395.0391, Y 54.6186, Z -4.6667, A 0.000, B 0.000, C 0.000 }
gfCNCPoint3[19591] = {X 395.7864, Y 53.9833, Z -4.6667, A 0.000, B 0.000, C 0.000 }
gfCNCPoint3[19592] = {X 396.6455, Y 53.5102, Z -4.6667, A 0.000, B 0.000, C 0.000 }
gfCNCPoint3[19593] = {X 397.5819, Y 53.2186, Z -4.6667, A 0.000, B 0.000, C 0.000 }
gfCNCPoint3[19594] = {X 398.5577, Y 53.1200, Z -4.6667, A 0.000, B 0.000, C 0.000 }
gfCNCPoint3[19595] = {X 419.4886, Y 53.1200, Z -4.6667, A 0.000, B 0.000, C 0.000 }
gfCNCPoint3[19596] = {X 420.5534, Y 53.2376, Z -4.6667, A 0.000, B 0.000, C 0.000 }
gfCNCPoint3[19597] = {X 421.5668, Y 53.5847, Z -4.6667, A 0.000, B 0.000, C 0.000 }
gfCNCPoint3[19598] = {X 422.4802, Y 54.1445, Z -4.6667, A 0.000, B 0.000, C 0.000 }
gfCNCPoint3[19599] = {X 423.2493, Y 54.8901, Z -4.6667, A 0.000, B 0.000, C 0.000 }
gfCNCPoint3[19600] = {X 423.8373, Y 55.7856, Z -4.6667, A 0.000, B 0.000, C 0.000 }
gfCNCPoint3[19601] = {X 424.2157, Y 56.7878, Z -4.6667, A 0.000, B 0.000, C 0.000 }
gfCNCPoint3[19602] = {X 424.3662, Y 57.8484, Z -4.6667, A 0.000, B 0.000, C 0.000 }
gfCNCPoint3[19603] = {X 429.8190, Y 59.9732, Z -4.6667, A 0.000, B 0.000, C 0.000 }
gfCNCPoint3[19604] = {X 457.2986, Y 70.8760, Z -4.6667, A 0.000, B 0.000, C 0.000 }
gfCNCPoint3[19605] = {X 457.2990, Y 63.6740, Z -4.6667, A 0.000, B 0.000, C 0.000 }
gfCNCPoint3[19606] = {X 456.2908, Y 63.3057, Z -4.6667, A 0.000, B 0.000, C 0.000 }
gfCNCPoint3[19607] = {X 455.3876, Y 62.7258, Z -4.6667, A 0.000, B 0.000, C 0.000 }
gfCNCPoint3[19608] = {X 454.6329, Y 61.9624, Z -4.6667, A 0.000, B 0.000, C 0.000 }
gfCNCPoint3[19609] = {X 454.0634, Y 61.0526, Z -4.6667, A 0.000, B 0.000, C 0.000 }
gfCNCPoint3[19610] = {X 453.7066, Y 60.0402, Z -4.6667, A 0.000, B 0.000, C 0.000 }
gfCNCPoint3[19611] = {X 453.5798, Y 58.9744, Z -4.6667, A 0.000, B 0.000, C 0.000 }
gfCNCPoint3[19612] = {X 453.5796, Y 58.0000, Z -4.6667, A 0.000, B 0.000, C 0.000 }
gfCNCPoint3[19613] = {X 453.6734, Y 57.0480, Z -4.6667, A 0.000, B 0.000, C 0.000 }
gfCNCPoint3[19614] = {X 453.9511, Y 56.1325, Z -4.6667, A 0.000, B 0.000, C 0.000 }
gfCNCPoint3[19615] = {X 454.4020, Y 55.2888, Z -4.6667, A 0.000, B 0.000, C 0.000 }
gfCNCPoint3[19616] = {X 455.0089, Y 54.5493, Z -4.6667, A 0.000, B 0.000, C 0.000 }
gfCNCPoint3[19617] = {X 455.7484, Y 53.9424, Z -4.6667, A 0.000, B 0.000, C 0.000 }
gfCNCPoint3[19618] = {X 456.5921, Y 53.4915, Z -4.6667, A 0.000, B 0.000, C 0.000 }
gfCNCPoint3[19619] = {X 457.5076, Y 53.2138, Z -4.6667, A 0.000, B 0.000, C 0.000 }
gfCNCPoint3[19620] = {X 458.4596, Y 53.1200, Z -4.6667, A 0.000, B 0.000, C 0.000 }
gfCNCPoint3[19621] = {X 475.0000, Y 53.1200, Z -4.6667, A 0.000, B 0.000, C 0.000 }
gfCNCPoint3[19622] = {X 475.9520, Y 53.2138, Z -4.6667, A 0.000, B 0.000, C 0.000 }
gfCNCPoint3[19623] = {X 476.8675, Y 53.4915, Z -4.6667, A 0.000, B 0.000, C 0.000 }
gfCNCPoint3[19624] = {X 477.7112, Y 53.9424, Z -4.6667, A 0.000, B 0.000, C 0.000 }
gfCNCPoint3[19625] = {X 478.4507, Y 54.5493, Z -4.6667, A 0.000, B 0.000, C 0.000 }
gfCNCPoint3[19626] = {X 479.0576, Y 55.2888, Z -4.6667, A 0.000, B 0.000, C 0.000 }
gfCNCPoint3[19627] = {X 479.5085, Y 56.1325, Z -4.6667, A 0.000, B 0.000, C 0.000 }
gfCNCPoint3[19628] = {X 479.7862, Y 57.0480, Z -4.6667, A 0.000, B 0.000, C 0.000 }
gfCNCPoint3[19629] = {X 479.8800, Y 58.0000, Z -4.6667, A 0.000, B 0.000, C 0.000 }
gfCNCPoint3[19630] = {X 479.8798, Y 58.9744, Z -4.6667, A 0.000, B 0.000, C 0.000 }
gfCNCPoint3[19631] = {X 479.7530, Y 60.0403, Z -4.6667, A 0.000, B 0.000, C 0.000 }
gfCNCPoint3[19632] = {X 479.3961, Y 61.0527, Z -4.6667, A 0.000, B 0.000, C 0.000 }
gfCNCPoint3[19633] = {X 478.8266, Y 61.9626, Z -4.6667, A 0.000, B 0.000, C 0.000 }
gfCNCPoint3[19634] = {X 478.0718, Y 62.7259, Z -4.6667, A 0.000, B 0.000, C 0.000 }
gfCNCPoint3[19635] = {X 477.1685, Y 63.3058, Z -4.6667, A 0.000, B 0.000, C 0.000 }
gfCNCPoint3[19636] = {X 476.1602, Y 63.6741, Z -4.6667, A 0.000, B 0.000, C 0.000 }
gfCNCPoint3[19637] = {X 476.1607, Y 92.3315, Z -4.6667, A 0.000, B 0.000, C 0.000 }
gfCNCPoint3[19638] = {X 476.3640, Y 92.3910, Z -4.6667, A 0.000, B 0.000, C 0.000 }
gfCNCPoint3[19639] = {X 476.5657, Y 92.4557, Z -4.6667, A 0.000, B 0.000, C 0.000 }
gfCNCPoint3[19640] = {X 477.4831, Y 92.8727, Z -4.6667, A 0.000, B 0.000, C 0.000 }
gfCNCPoint3[19641] = {X 478.2946, Y 93.4702, Z -4.6667, A 0.000, B 0.000, C 0.000 }
gfCNCPoint3[19642] = {X 478.9652, Y 94.2224, Z -4.6667, A 0.000, B 0.000, C 0.000 }
gfCNCPoint3[19643] = {X 479.4660, Y 95.0968, Z -4.6667, A 0.000, B 0.000, C 0.000 }
gfCNCPoint3[19644] = {X 479.7754, Y 96.0559, Z -4.6667, A 0.000, B 0.000, C 0.000 }
gfCNCPoint3[19645] = {X 479.8800, Y 97.0582, Z -4.6667, A 0.000, B 0.000, C 0.000 }
gfCNCPoint3[19646] = {X 479.8800, Y 97.6950, Z -4.6667, A 0.000, B 0.000, C 0.000 }
gfCNCPoint3[19647] = {X 479.4000, Y 97.6950, Z -4.6667, A 0.000, B 0.000, C 0.000 }
gfCNCPoint3[19648] = {X 479.4000, Y 98.0000, Z -4.6667, A 0.000, B 0.000, C 0.000 }
gfCNCPoint3[19649] = {X 479.2897, Y 98.9791, Z -4.6667, A 0.000, B 0.000, C 0.000 }
gfCNCPoint3[19650] = {X 478.9643, Y 99.9091, Z -4.6667, A 0.000, B 0.000, C 0.000 }
gfCNCPoint3[19651] = {X 478.4401, Y 100.7434, Z -4.6667, A 0.000, B 0.000, C 0.000 }
gfCNCPoint3[19652] = {X 477.7434, Y 101.4401, Z -4.6667, A 0.000, B 0.000, C 0.000 }
gfCNCPoint3[19653] = {X 476.9091, Y 101.9643, Z -4.6667, A 0.000, B 0.000, C 0.000 }
gfCNCPoint3[19654] = {X 475.9791, Y 102.2897, Z -4.6667, A 0.000, B 0.000, C 0.000 }
gfCNCPoint3[19655] = {X 475.0000, Y 102.4000, Z -4.6667, A 0.000, B 0.000, C 0.000 }
gfCNCPoint3[19656] = {X 458.4596, Y 102.4000, Z -4.6667, A 0.000, B 0.000, C 0.000 }
gfCNCPoint3[19657] = {X 457.4805, Y 102.2897, Z -4.6667, A 0.000, B 0.000, C 0.000 }
gfCNCPoint3[19658] = {X 456.5505, Y 101.9643, Z -4.6667, A 0.000, B 0.000, C 0.000 }
gfCNCPoint3[19659] = {X 455.7162, Y 101.4401, Z -4.6667, A 0.000, B 0.000, C 0.000 }
gfCNCPoint3[19660] = {X 455.0195, Y 100.7434, Z -4.6667, A 0.000, B 0.000, C 0.000 }
gfCNCPoint3[19661] = {X 454.4953, Y 99.9091, Z -4.6667, A 0.000, B 0.000, C 0.000 }
gfCNCPoint3[19662] = {X 454.1699, Y 98.9791, Z -4.6667, A 0.000, B 0.000, C 0.000 }
gfCNCPoint3[19663] = {X 454.0596, Y 98.0000, Z -4.6667, A 0.000, B 0.000, C 0.000 }
gfCNCPoint3[19664] = {X 454.0596, Y 97.0659, Z -4.6667, A 0.000, B 0.000, C 0.000 }
gfCNCPoint3[19665] = {X 454.1492, Y 96.1826, Z -4.6667, A 0.000, B 0.000, C 0.000 }
gfCNCPoint3[19666] = {X 454.4143, Y 95.3353, Z -4.6667, A 0.000, B 0.000, C 0.000 }
gfCNCPoint3[19667] = {X 454.8440, Y 94.5584, Z -4.6667, A 0.000, B 0.000, C 0.000 }
gfCNCPoint3[19668] = {X 455.4210, Y 93.8836, Z -4.6667, A 0.000, B 0.000, C 0.000 }
gfCNCPoint3[19669] = {X 456.1217, Y 93.3384, Z -4.6667, A 0.000, B 0.000, C 0.000 }
gfCNCPoint3[19670] = {X 456.9176, Y 92.9450, Z -4.6667, A 0.000, B 0.000, C 0.000 }
gfCNCPoint3[19671] = {X 457.7763, Y 92.7193, Z -4.6667, A 0.000, B 0.000, C 0.000 }
gfCNCPoint3[19672] = {X 457.7763, Y 85.6495, Z -4.6667, A 0.000, B 0.000, C 0.000 }
gfCNCPoint3[19673] = {X 444.8682, Y 80.5895, Z -4.6667, A 0.000, B 0.000, C 0.000 }
gfCNCPoint3[19674] = {X 420.1038, Y 96.6316, Z -4.6667, A 0.000, B 0.000, C 0.000 }
gfCNCPoint3[19675] = {X 420.1067, Y 97.0659, Z -4.6667, A 0.000, B 0.000, C 0.000 }
gfCNCPoint3[19676] = {X 420.1067, Y 98.0000, Z -4.6667, A 0.000, B 0.000, C 0.000 }
gfCNCPoint3[19677] = {X 419.9964, Y 98.9791, Z -4.6667, A 0.000, B 0.000, C 0.000 }
gfCNCPoint3[19678] = {X 419.6710, Y 99.9091, Z -4.6667, A 0.000, B 0.000, C 0.000 }
gfCNCPoint3[19679] = {X 419.1468, Y 100.7434, Z -4.6667, A 0.000, B 0.000, C 0.000 }
gfCNCPoint3[19680] = {X 418.4501, Y 101.4401, Z -4.6667, A 0.000, B 0.000, C 0.000 }
gfCNCPoint3[19681] = {X 417.6158, Y 101.9643, Z -4.6667, A 0.000, B 0.000, C 0.000 }
gfCNCPoint3[19682] = {X 416.6858, Y 102.2897, Z -4.6667, A 0.000, B 0.000, C 0.000 }
gfCNCPoint3[19683] = {X 415.7067, Y 102.4000, Z -4.6667, A 0.000, B 0.000, C 0.000 }
gfCNCPoint3[19684] = {X 396.4059, Y 102.4000, Z -4.6667, A 0.000, B 0.000, C 0.000 }
gfCNCPoint3[19685] = {X 395.4269, Y 102.2897, Z -4.6667, A 0.000, B 0.000, C 0.000 }
gfCNCPoint3[19686] = {X 394.4969, Y 101.9643, Z -4.6667, A 0.000, B 0.000, C 0.000 }
gfCNCPoint3[19687] = {X 393.6626, Y 101.4401, Z -4.6667, A 0.000, B 0.000, C 0.000 }
gfCNCPoint3[19688] = {X 392.9659, Y 100.7434, Z -4.6667, A 0.000, B 0.000, C 0.000 }
gfCNCPoint3[19689] = {X 392.4417, Y 99.9091, Z -4.6667, A 0.000, B 0.000, C 0.000 }
gfCNCPoint3[19690] = {X 392.1163, Y 98.9791, Z -4.6667, A 0.000, B 0.000, C 0.000 }
gfCNCPoint3[19691] = {X 392.0059, Y 98.0000, Z -4.6667, A 0.000, B 0.000, C 0.000 }
gfCNCPoint3[19692] = {X 392.0059, Y 97.0659, Z -4.6667, A 0.000, B 0.000, C 0.000 }
gfCNCPoint3[19693] = {X 392.1171, Y 96.0834, Z -4.6667, A 0.000, B 0.000, C 0.000 }
gfCNCPoint3[19694] = {X 392.4448, Y 95.1504, Z -4.6667, A 0.000, B 0.000, C 0.000 }
gfCNCPoint3[19695] = {X 392.9725, Y 94.3143, Z -4.6667, A 0.000, B 0.000, C 0.000 }
gfCNCPoint3[19696] = {X 393.6737, Y 93.6170, Z -4.6667, A 0.000, B 0.000, C 0.000 }
gfCNCPoint3[19697] = {X 394.5129, Y 93.0940, Z -4.6667, A 0.000, B 0.000, C 0.000 }
gfCNCPoint3[19698] = {X 395.4477, Y 92.7716, Z -4.6667, A 0.000, B 0.000, C 0.000 }
gfCNCPoint3[19699] = {X 396.4308, Y 92.6660, Z -4.6667, A 0.000, B 0.000, C 0.000 }
gfCNCPoint3[19700] = {X 397.3589, Y 92.6230, Z -4.6667, A 0.000, B 0.000, C 0.000 }
gfCNCPoint3[19701] = {X 398.2838, Y 92.5349, Z -4.6667, A 0.000, B 0.000, C 0.000 }
gfCNCPoint3[19702] = {X 398.9171, Y 92.3812, Z -4.6667, A 0.000, B 0.000, C 0.000 }
gfCNCPoint3[19703] = {X 399.5003, Y 92.0904, Z -4.6667, A 0.000, B 0.000, C 0.000 }
gfCNCPoint3[19704] = {X 405.1767, Y 88.4328, Z -4.6667, A 0.000, B 0.000, C 0.000 }
gfCNCPoint3[19705] = {X 427.8788, Y 73.9165, Z -4.6667, A 0.000, B 0.000, C 0.000 }
gfCNCPoint3[19706] = {X 403.7262, Y 64.4403, Z -4.6667, A 0.000, B 0.000, C 0.000 }
gfCNCPoint3[19707] = {X 402.0392, Y 63.8817, Z -4.6667, A 0.000, B 0.000, C 0.000 }
gfCNCPoint3[19708] = {X 400.3010, Y 63.5114, Z -4.6667, A 0.000, B 0.000, C 0.000 }
gfCNCPoint3[19709] = {X 398.5328, Y 63.3340, Z -4.6667, A 0.000, B 0.000, C 0.000 }
gfCNCPoint3[19710] = {X 397.5578, Y 63.2189, Z -4.6667, A 0.000, B 0.000, C 0.000 }
gfCNCPoint3[19711] = {X 396.6326, Y 62.8906, Z -4.6667, A 0.000, B 0.000, C 0.000 }
gfCNCPoint3[19712] = {X 395.8032, Y 62.3652, Z -4.6667, A 0.000, B 0.000, C 0.000 }
gfCNCPoint3[19713] = {X 395.1110, Y 61.6691, Z -4.6667, A 0.000, B 0.000, C 0.000 }
gfCNCPoint3[19714] = {X 394.5904, Y 60.8367, Z -4.6667, A 0.000, B 0.000, C 0.000 }
gfCNCPoint3[19715] = {X 394.2672, Y 59.9097, Z -4.6667, A 0.000, B 0.000, C 0.000 }
gfCNCPoint3[19716] = {X 394.1577, Y 58.9341, Z -4.6667, A 0.000, B 0.000, C 0.000 }
gfCNCPoint3[19717] = {X 394.1577, Y 58.0000, Z -4.6667, A 0.000, B 0.000, C 0.000 }
gfCNCPoint3[19718] = {X 394.2680, Y 57.0209, Z -4.6667, A 0.000, B 0.000, C 0.000 }
gfCNCPoint3[19719] = {X 394.5935, Y 56.0909, Z -4.6667, A 0.000, B 0.000, C 0.000 }
gfCNCPoint3[19720] = {X 395.1177, Y 55.2566, Z -4.6667, A 0.000, B 0.000, C 0.000 }
gfCNCPoint3[19721] = {X 395.8144, Y 54.5599, Z -4.6667, A 0.000, B 0.000, C 0.000 }
gfCNCPoint3[19722] = {X 396.6486, Y 54.0357, Z -4.6667, A 0.000, B 0.000, C 0.000 }
gfCNCPoint3[19723] = {X 397.5786, Y 53.7103, Z -4.6667, A 0.000, B 0.000, C 0.000 }
gfCNCPoint3[19724] = {X 398.5577, Y 53.6000, Z -4.6667, A 0.000, B 0.000, C 0.000 }
gfCNCPoint3[19725] = {X 419.4886, Y 53.6000, Z -4.6667, A 0.000, B 0.000, C 0.000 }
gfCNCPoint3[19726] = {X 420.4677, Y 53.7103, Z -4.6667, A 0.000, B 0.000, C 0.000 }
gfCNCPoint3[19727] = {X 421.3977, Y 54.0357, Z -4.6667, A 0.000, B 0.000, C 0.000 }
gfCNCPoint3[19728] = {X 422.2320, Y 54.5599, Z -4.6667, A 0.000, B 0.000, C 0.000 }
gfCNCPoint3[19729] = {X 422.9287, Y 55.2566, Z -4.6667, A 0.000, B 0.000, C 0.000 }
gfCNCPoint3[19730] = {X 423.4529, Y 56.0909, Z -4.6667, A 0.000, B 0.000, C 0.000 }
gfCNCPoint3[19731] = {X 423.7783, Y 57.0209, Z -4.6667, A 0.000, B 0.000, C 0.000 }
gfCNCPoint3[19732] = {X 423.8886, Y 58.0000, Z -4.6667, A 0.000, B 0.000, C 0.000 }
gfCNCPoint3[19733] = {X 423.8886, Y 58.1775, Z -4.6667, A 0.000, B 0.000, C 0.000 }
gfCNCPoint3[19734] = {X 429.6420, Y 60.4194, Z -4.6667, A 0.000, B 0.000, C 0.000 }
gfCNCPoint3[19735] = {X 457.7786, Y 71.5828, Z -4.6667, A 0.000, B 0.000, C 0.000 }
gfCNCPoint3[19736] = {X 457.7790, Y 63.2811, Z -4.6667, A 0.000, B 0.000, C 0.000 }
gfCNCPoint3[19737] = {X 456.9199, Y 63.0559, Z -4.6667, A 0.000, B 0.000, C 0.000 }
gfCNCPoint3[19738] = {X 456.1234, Y 62.6626, Z -4.6667, A 0.000, B 0.000, C 0.000 }
gfCNCPoint3[19739] = {X 455.4222, Y 62.1175, Z -4.6667, A 0.000, B 0.000, C 0.000 }
gfCNCPoint3[19740] = {X 454.8447, Y 61.4426, Z -4.6667, A 0.000, B 0.000, C 0.000 }
gfCNCPoint3[19741] = {X 454.4146, Y 60.6654, Z -4.6667, A 0.000, B 0.000, C 0.000 }
gfCNCPoint3[19742] = {X 454.1493, Y 59.8177, Z -4.6667, A 0.000, B 0.000, C 0.000 }
gfCNCPoint3[19743] = {X 454.0596, Y 58.9341, Z -4.6667, A 0.000, B 0.000, C 0.000 }
gfCNCPoint3[19744] = {X 454.0596, Y 58.0000, Z -4.6667, A 0.000, B 0.000, C 0.000 }
gfCNCPoint3[19745] = {X 454.1699, Y 57.0209, Z -4.6667, A 0.000, B 0.000, C 0.000 }
gfCNCPoint3[19746] = {X 454.4953, Y 56.0909, Z -4.6667, A 0.000, B 0.000, C 0.000 }
gfCNCPoint3[19747] = {X 455.0195, Y 55.2566, Z -4.6667, A 0.000, B 0.000, C 0.000 }
gfCNCPoint3[19748] = {X 455.7162, Y 54.5599, Z -4.6667, A 0.000, B 0.000, C 0.000 }
gfCNCPoint3[19749] = {X 456.5505, Y 54.0357, Z -4.6667, A 0.000, B 0.000, C 0.000 }
gfCNCPoint3[19750] = {X 457.4805, Y 53.7103, Z -4.6667, A 0.000, B 0.000, C 0.000 }
gfCNCPoint3[19751] = {X 458.4596, Y 53.6000, Z -4.6667, A 0.000, B 0.000, C 0.000 }
gfCNCPoint3[19752] = {X 475.0000, Y 53.6000, Z -4.6667, A 0.000, B 0.000, C 0.000 }
gfCNCPoint3[19753] = {X 475.9791, Y 53.7103, Z -4.6667, A 0.000, B 0.000, C 0.000 }
gfCNCPoint3[19754] = {X 476.9091, Y 54.0357, Z -4.6667, A 0.000, B 0.000, C 0.000 }
gfCNCPoint3[19755] = {X 477.7434, Y 54.5599, Z -4.6667, A 0.000, B 0.000, C 0.000 }
gfCNCPoint3[19756] = {X 478.4401, Y 55.2566, Z -4.6667, A 0.000, B 0.000, C 0.000 }
gfCNCPoint3[19757] = {X 478.9643, Y 56.0909, Z -4.6667, A 0.000, B 0.000, C 0.000 }
gfCNCPoint3[19758] = {X 479.2897, Y 57.0209, Z -4.6667, A 0.000, B 0.000, C 0.000 }
gfCNCPoint3[19759] = {X 479.4000, Y 58.0000, Z -4.6667, A 0.000, B 0.000, C 0.000 }
gfCNCPoint3[19760] = {X 479.3998, Y 58.9704, Z -4.6667, A 0.000, B 0.000, C 0.000 }
gfCNCPoint3[19761] = {X 479.3040, Y 59.8483, Z -4.6667, A 0.000, B 0.000, C 0.000 }
gfCNCPoint3[19762] = {X 479.0347, Y 60.6894, Z -4.6667, A 0.000, B 0.000, C 0.000 }
gfCNCPoint3[19763] = {X 478.6029, Y 61.4597, Z -4.6667, A 0.000, B 0.000, C 0.000 }
gfCNCPoint3[19764] = {X 478.0260, Y 62.1283, Z -4.6667, A 0.000, B 0.000, C 0.000 }
gfCNCPoint3[19765] = {X 477.3272, Y 62.6683, Z -4.6667, A 0.000, B 0.000, C 0.000 }
gfCNCPoint3[19766] = {X 476.5346, Y 63.0578, Z -4.6667, A 0.000, B 0.000, C 0.000 }
gfCNCPoint3[19767] = {X 475.6802, Y 63.2812, Z -4.6667, A 0.000, B 0.000, C 0.000 }
gfCNCPoint3[19768] = {X 475.6807, Y 92.7042, Z -4.6667, A 0.000, B 0.000, C 0.000 }
gfCNCPoint3[19769] = {X 476.0496, Y 92.7988, Z -4.6667, A 0.000, B 0.000, C 0.000 }
gfCNCPoint3[19770] = {X 476.4135, Y 92.9109, Z -4.6667, A 0.000, B 0.000, C 0.000 }
gfCNCPoint3[19771] = {X 477.2402, Y 93.2867, Z -4.6667, A 0.000, B 0.000, C 0.000 }
gfCNCPoint3[19772] = {X 477.9714, Y 93.8250, Z -4.6667, A 0.000, B 0.000, C 0.000 }
gfCNCPoint3[19773] = {X 478.5757, Y 94.5029, Z -4.6667, A 0.000, B 0.000, C 0.000 }
gfCNCPoint3[19774] = {X 479.0269, Y 95.2908, Z -4.6667, A 0.000, B 0.000, C 0.000 }
gfCNCPoint3[19775] = {X 479.3057, Y 96.1550, Z -4.6667, A 0.000, B 0.000, C 0.000 }
gfCNCPoint3[19776] = {X 479.4000, Y 97.0582, Z -4.6667, A 0.000, B 0.000, C 0.000 }
gfCNCPoint3[19777] = {X 479.4000, Y 97.6950, Z -4.6667, A 0.000, B 0.000, C 0.000 }
gfCNCPoint3[19778] = {X 479.8800, Y 97.6950, Z -4.6667, A 0.000, B 0.000, C 0.000 }
gfCNCPoint3[19779] = {X 507.6815, Y 97.6950, Z -4.6667, A 0.000, B 0.000, C 0.000 }
gfCNCPoint3[19780] = {X 507.6815, Y 100.0950, Z -4.6667, A 0.000, B 0.000, C 0.000 }
gfCNCPoint3[19781] = {X 600.0148, Y 100.0950, Z -4.6667, A 0.000, B 0.000, C 0.000 }
gfCNCPoint3[19782] = {X 600.0672, Y 100.0698, Z -4.6667, A 0.000, B 0.000, C 0.000 }
gfCNCPoint3[19783] = {X 600.0949, Y 100.0187, Z -4.6667, A 0.000, B 0.000, C 0.000 }
gfCNCPoint3[19784] = {X 600.0966, Y 99.1432, Z -4.6667, A 0.000, B 0.000, C 0.000 }
gfCNCPoint3[19785] = {X 600.0966, Y 49.8790, Z -4.6667, A 0.000, B 0.000, C 0.000 }
gfCNCPoint3[19786] = {X 601.1112, Y 49.7518, Z -4.6667, A 0.000, B 0.000, C 0.000 }
gfCNCPoint3[19787] = {X 602.0769, Y 49.4160, Z -4.6667, A 0.000, B 0.000, C 0.000 }
gfCNCPoint3[19788] = {X 602.9516, Y 48.8862, Z -4.6667, A 0.000, B 0.000, C 0.000 }
gfCNCPoint3[19789] = {X 603.6966, Y 48.1859, Z -4.6667, A 0.000, B 0.000, C 0.000 }
gfCNCPoint3[19790] = {X 603.6966, Y 47.3865, Z -4.6667, A 0.000, B 0.000, C 0.000 }
gfCNCPoint3[19791] = {X 603.1503, Y 48.0718, Z -4.6667, A 0.000, B 0.000, C 0.000 }
gfCNCPoint3[19792] = {X 602.4790, Y 48.6352, Z -4.6667, A 0.000, B 0.000, C 0.000 }
gfCNCPoint3[19793] = {X 601.7094, Y 49.0544, Z -4.6667, A 0.000, B 0.000, C 0.000 }
gfCNCPoint3[19794] = {X 600.8720, Y 49.3127, Z -4.6667, A 0.000, B 0.000, C 0.000 }
gfCNCPoint3[19795] = {X 600.0000, Y 49.4000, Z -4.6667, A 0.000, B 0.000, C 0.000 }
gfCNCPoint3[19796] = {X 593.5565, Y 49.4000, Z -4.6667, A 0.000, B 0.000, C 0.000 }
gfCNCPoint3[19797] = {X 592.5988, Y 49.2945, Z -4.6667, A 0.000, B 0.000, C 0.000 }
gfCNCPoint3[19798] = {X 591.6870, Y 48.9831, Z -4.6667, A 0.000, B 0.000, C 0.000 }
gfCNCPoint3[19799] = {X 590.8648, Y 48.4806, Z -4.6667, A 0.000, B 0.000, C 0.000 }
gfCNCPoint3[19800] = {X 590.1717, Y 47.8112, Z -4.6667, A 0.000, B 0.000, C 0.000 }
gfCNCPoint3[19801] = {X 589.6410, Y 47.0071, Z -4.6667, A 0.000, B 0.000, C 0.000 }
gfCNCPoint3[19802] = {X 589.3741, Y 46.3664, Z -4.6667, A 0.000, B 0.000, C 0.000 }
gfCNCPoint3[19803] = {X 589.2113, Y 45.6918, Z -4.6667, A 0.000, B 0.000, C 0.000 }
gfCNCPoint3[19804] = {X 589.1565, Y 45.0000, Z -4.6667, A 0.000, B 0.000, C 0.000 }
gfCNCPoint3[19805] = {X 589.1565, Y 44.0642, Z -4.6667, A 0.000, B 0.000, C 0.000 }
gfCNCPoint3[19806] = {X 589.2608, Y 43.1278, Z -4.6667, A 0.000, B 0.000, C 0.000 }
gfCNCPoint3[19807] = {X 589.5602, Y 42.2344, Z -4.6667, A 0.000, B 0.000, C 0.000 }
gfCNCPoint3[19808] = {X 590.0414, Y 41.4244, Z -4.6667, A 0.000, B 0.000, C 0.000 }
gfCNCPoint3[19809] = {X 590.6827, Y 40.7341, Z -4.6667, A 0.000, B 0.000, C 0.000 }
gfCNCPoint3[19810] = {X 590.6841, Y 40.3069, Z -4.6667, A 0.000, B 0.000, C 0.000 }
gfCNCPoint3[19811] = {X 590.6833, Y 35.2182, Z -4.6667, A 0.000, B 0.000, C 0.000 }
gfCNCPoint3[19812] = {X 590.6831, Y 33.9406, Z -4.6667, A 0.000, B 0.000, C 0.000 }
gfCNCPoint3[19813] = {X 585.5192, Y 46.6830, Z -4.6667, A 0.000, B 0.000, C 0.000 }
gfCNCPoint3[19814] = {X 585.4476, Y 46.8466, Z -4.6667, A 0.000, B 0.000, C 0.000 }
gfCNCPoint3[19815] = {X 585.3694, Y 47.0071, Z -4.6667, A 0.000, B 0.000, C 0.000 }
gfCNCPoint3[19816] = {X 584.8417, Y 47.8075, Z -4.6667, A 0.000, B 0.000, C 0.000 }
gfCNCPoint3[19817] = {X 584.1532, Y 48.4747, Z -4.6667, A 0.000, B 0.000, C 0.000 }
gfCNCPoint3[19818] = {X 583.3365, Y 48.9769, Z -4.6667, A 0.000, B 0.000, C 0.000 }
gfCNCPoint3[19819] = {X 582.4111, Y 49.2946, Z -4.6667, A 0.000, B 0.000, C 0.000 }
gfCNCPoint3[19820] = {X 581.4384, Y 49.4000, Z -4.6667, A 0.000, B 0.000, C 0.000 }
gfCNCPoint3[19821] = {X 580.4664, Y 49.2878, Z -4.6667, A 0.000, B 0.000, C 0.000 }
gfCNCPoint3[19822] = {X 579.5433, Y 48.9635, Z -4.6667, A 0.000, B 0.000, C 0.000 }
gfCNCPoint3[19823] = {X 578.7146, Y 48.4433, Z -4.6667, A 0.000, B 0.000, C 0.000 }
gfCNCPoint3[19824] = {X 578.0214, Y 47.7529, Z -4.6667, A 0.000, B 0.000, C 0.000 }
gfCNCPoint3[19825] = {X 577.4979, Y 46.9263, Z -4.6667, A 0.000, B 0.000, C 0.000 }
gfCNCPoint3[19826] = {X 577.4375, Y 46.7968, Z -4.6667, A 0.000, B 0.000, C 0.000 }
gfCNCPoint3[19827] = {X 577.3813, Y 46.6655, Z -4.6667, A 0.000, B 0.000, C 0.000 }
gfCNCPoint3[19828] = {X 572.0989, Y 33.7486, Z -4.6667, A 0.000, B 0.000, C 0.000 }
gfCNCPoint3[19829] = {X 572.0992, Y 40.7332, Z -4.6667, A 0.000, B 0.000, C 0.000 }
gfCNCPoint3[19830] = {X 572.7437, Y 41.4223, Z -4.6667, A 0.000, B 0.000, C 0.000 }
gfCNCPoint3[19831] = {X 573.2265, Y 42.2330, Z -4.6667, A 0.000, B 0.000, C 0.000 }
gfCNCPoint3[19832] = {X 573.5253, Y 43.1279, Z -4.6667, A 0.000, B 0.000, C 0.000 }
gfCNCPoint3[19833] = {X 573.6264, Y 44.0660, Z -4.6667, A 0.000, B 0.000, C 0.000 }
gfCNCPoint3[19834] = {X 573.6264, Y 45.0000, Z -4.6667, A 0.000, B 0.000, C 0.000 }
gfCNCPoint3[19835] = {X 573.5140, Y 45.9884, Z -4.6667, A 0.000, B 0.000, C 0.000 }
gfCNCPoint3[19836] = {X 573.1824, Y 46.9263, Z -4.6667, A 0.000, B 0.000, C 0.000 }
gfCNCPoint3[19837] = {X 572.6569, Y 47.7553, Z -4.6667, A 0.000, B 0.000, C 0.000 }
gfCNCPoint3[19838] = {X 571.9608, Y 48.4472, Z -4.6667, A 0.000, B 0.000, C 0.000 }
gfCNCPoint3[19839] = {X 571.1286, Y 48.9676, Z -4.6667, A 0.000, B 0.000, C 0.000 }
gfCNCPoint3[19840] = {X 570.2018, Y 49.2905, Z -4.6667, A 0.000, B 0.000, C 0.000 }
gfCNCPoint3[19841] = {X 569.2264, Y 49.4000, Z -4.6667, A 0.000, B 0.000, C 0.000 }
gfCNCPoint3[19842] = {X 562.4443, Y 49.4000, Z -4.6667, A 0.000, B 0.000, C 0.000 }
gfCNCPoint3[19843] = {X 561.4652, Y 49.2897, Z -4.6667, A 0.000, B 0.000, C 0.000 }
gfCNCPoint3[19844] = {X 560.5352, Y 48.9643, Z -4.6667, A 0.000, B 0.000, C 0.000 }
gfCNCPoint3[19845] = {X 559.7009, Y 48.4401, Z -4.6667, A 0.000, B 0.000, C 0.000 }
gfCNCPoint3[19846] = {X 559.0042, Y 47.7434, Z -4.6667, A 0.000, B 0.000, C 0.000 }
gfCNCPoint3[19847] = {X 558.4800, Y 46.9091, Z -4.6667, A 0.000, B 0.000, C 0.000 }
gfCNCPoint3[19848] = {X 558.1546, Y 45.9791, Z -4.6667, A 0.000, B 0.000, C 0.000 }
gfCNCPoint3[19849] = {X 558.0443, Y 45.0000, Z -4.6667, A 0.000, B 0.000, C 0.000 }
gfCNCPoint3[19850] = {X 558.0443, Y 44.0643, Z -4.6667, A 0.000, B 0.000, C 0.000 }
gfCNCPoint3[19851] = {X 558.1483, Y 43.1277, Z -4.6667, A 0.000, B 0.000, C 0.000 }
gfCNCPoint3[19852] = {X 558.4480, Y 42.2341, Z -4.6667, A 0.000, B 0.000, C 0.000 }
gfCNCPoint3[19853] = {X 558.9297, Y 41.4241, Z -4.6667, A 0.000, B 0.000, C 0.000 }
gfCNCPoint3[19854] = {X 559.5718, Y 40.7342, Z -4.6667, A 0.000, B 0.000, C 0.000 }
gfCNCPoint3[19855] = {X 559.5718, Y 9.2670, Z -4.6667, A 0.000, B 0.000, C 0.000 }
gfCNCPoint3[19856] = {X 558.9272, Y 8.5779, Z -4.6667, A 0.000, B 0.000, C 0.000 }
gfCNCPoint3[19857] = {X 558.4443, Y 7.7672, Z -4.6667, A 0.000, B 0.000, C 0.000 }
gfCNCPoint3[19858] = {X 558.1455, Y 6.8721, Z -4.6667, A 0.000, B 0.000, C 0.000 }
gfCNCPoint3[19859] = {X 558.0443, Y 5.9340, Z -4.6667, A 0.000, B 0.000, C 0.000 }
gfCNCPoint3[19860] = {X 558.0443, Y 5.0000, Z -4.6667, A 0.000, B 0.000, C 0.000 }
gfCNCPoint3[19861] = {X 558.1353, Y 4.1097, Z -4.6667, A 0.000, B 0.000, C 0.000 }
gfCNCPoint3[19862] = {X 558.4046, Y 3.2562, Z -4.6667, A 0.000, B 0.000, C 0.000 }
gfCNCPoint3[19863] = {X 558.9155, Y 2.3717, Z -4.6667, A 0.000, B 0.000, C 0.000 }
gfCNCPoint3[19864] = {X 559.6166, Y 1.6289, Z -4.6667, A 0.000, B 0.000, C 0.000 }
gfCNCPoint3[19865] = {X 560.4700, Y 1.0678, Z -4.6667, A 0.000, B 0.000, C 0.000 }
gfCNCPoint3[19866] = {X 561.4298, Y 0.7185, Z -4.6667, A 0.000, B 0.000, C 0.000 }
gfCNCPoint3[19867] = {X 562.4443, Y 0.6000, Z -4.6667, A 0.000, B 0.000, C 0.000 }
gfCNCPoint3[19868] = {X 570.9376, Y 0.6000, Z -4.6667, A 0.000, B 0.000, C 0.000 }
gfCNCPoint3[19869] = {X 571.9520, Y 0.7185, Z -4.6667, A 0.000, B 0.000, C 0.000 }
gfCNCPoint3[19870] = {X 572.9118, Y 1.0678, Z -4.6667, A 0.000, B 0.000, C 0.000 }
gfCNCPoint3[19871] = {X 573.7653, Y 1.6289, Z -4.6667, A 0.000, B 0.000, C 0.000 }
gfCNCPoint3[19872] = {X 574.4663, Y 2.3717, Z -4.6667, A 0.000, B 0.000, C 0.000 }
gfCNCPoint3[19873] = {X 574.9772, Y 3.2562, Z -4.6667, A 0.000, B 0.000, C 0.000 }
gfCNCPoint3[19874] = {X 575.2317, Y 4.0407, Z -4.6667, A 0.000, B 0.000, C 0.000 }
gfCNCPoint3[19875] = {X 575.3353, Y 4.8589, Z -4.6667, A 0.000, B 0.000, C 0.000 }
gfCNCPoint3[19876] = {X 580.1328, Y 4.7050, Z -4.6667, A 0.000, B 0.000, C 0.000 }
gfCNCPoint3[19877] = {X 580.1364, Y 4.8525, Z -4.6667, A 0.000, B 0.000, C 0.000 }
gfCNCPoint3[19878] = {X 580.1376, Y 5.0000, Z -4.6667, A 0.000, B 0.000, C 0.000 }
gfCNCPoint3[19879] = {X 580.1376, Y 5.9338, Z -4.6667, A 0.000, B 0.000, C 0.000 }
gfCNCPoint3[19880] = {X 580.0685, Y 7.0588, Z -4.6667, A 0.000, B 0.000, C 0.000 }
gfCNCPoint3[19881] = {X 579.8625, Y 8.1668, Z -4.6667, A 0.000, B 0.000, C 0.000 }
gfCNCPoint3[19882] = {X 581.2004, Y 11.4525, Z -4.6667, A 0.000, B 0.000, C 0.000 }
gfCNCPoint3[19883] = {X 582.6184, Y 7.9846, Z -4.6667, A 0.000, B 0.000, C 0.000 }
gfCNCPoint3[19884] = {X 582.4489, Y 6.9995, Z -4.6667, A 0.000, B 0.000, C 0.000 }
gfCNCPoint3[19885] = {X 582.3872, Y 6.0018, Z -4.6667, A 0.000, B 0.000, C 0.000 }
gfCNCPoint3[19886] = {X 582.3870, Y 5.0000, Z -4.6667, A 0.000, B 0.000, C 0.000 }
gfCNCPoint3[19887] = {X 582.3881, Y 4.8525, Z -4.6667, A 0.000, B 0.000, C 0.000 }
gfCNCPoint3[19888] = {X 582.3917, Y 4.7050, Z -4.6667, A 0.000, B 0.000, C 0.000 }
gfCNCPoint3[19889] = {X 580.1328, Y 4.7050, Z -4.6667, A 0.000, B 0.000, C 0.000 }
gfCNCPoint3[19890] = {X 577.7341, Y 4.7819, Z -4.6667, A 0.000, B 0.000, C 0.000 }
gfCNCPoint3[19891] = {X 577.7367, Y 4.8910, Z -4.6667, A 0.000, B 0.000, C 0.000 }
gfCNCPoint3[19892] = {X 577.7376, Y 5.0000, Z -4.6667, A 0.000, B 0.000, C 0.000 }
gfCNCPoint3[19893] = {X 577.7376, Y 5.9339, Z -4.6667, A 0.000, B 0.000, C 0.000 }
gfCNCPoint3[19894] = {X 577.6318, Y 7.1286, Z -4.6667, A 0.000, B 0.000, C 0.000 }
gfCNCPoint3[19895] = {X 577.3178, Y 8.2861, Z -4.6667, A 0.000, B 0.000, C 0.000 }
gfCNCPoint3[19896] = {X 577.5057, Y 8.7428, Z -4.6667, A 0.000, B 0.000, C 0.000 }
gfCNCPoint3[19897] = {X 581.1958, Y 17.8052, Z -4.6667, A 0.000, B 0.000, C 0.000 }
gfCNCPoint3[19898] = {X 585.1515, Y 8.1307, Z -4.6667, A 0.000, B 0.000, C 0.000 }
gfCNCPoint3[19899] = {X 584.8835, Y 7.0757, Z -4.6667, A 0.000, B 0.000, C 0.000 }
gfCNCPoint3[19900] = {X 584.7872, Y 5.9914, Z -4.6667, A 0.000, B 0.000, C 0.000 }
gfCNCPoint3[19901] = {X 584.7870, Y 5.0000, Z -4.6667, A 0.000, B 0.000, C 0.000 }
gfCNCPoint3[19902] = {X 584.7878, Y 4.8910, Z -4.6667, A 0.000, B 0.000, C 0.000 }
gfCNCPoint3[19903] = {X 584.7905, Y 4.7819, Z -4.6667, A 0.000, B 0.000, C 0.000 }
gfCNCPoint3[19904] = {X 584.9505, Y 3.5174, Z -4.6667, A 0.000, B 0.000, C 0.000 }
gfCNCPoint3[19905] = {X 585.3438, Y 2.3050, Z -4.6667, A 0.000, B 0.000, C 0.000 }
gfCNCPoint3[19906] = {X 577.1807, Y 2.3050, Z -4.6667, A 0.000, B 0.000, C 0.000 }
gfCNCPoint3[19907] = {X 577.5740, Y 3.5174, Z -4.6667, A 0.000, B 0.000, C 0.000 }
gfCNCPoint3[19908] = {X 577.7341, Y 4.7819, Z -4.6667, A 0.000, B 0.000, C 0.000 }
gfCNCPoint3[19909] = {X 575.3353, Y 4.8589, Z -4.6667, A 0.000, B 0.000, C 0.000 }
gfCNCPoint3[19910] = {X 575.3370, Y 4.9294, Z -4.6667, A 0.000, B 0.000, C 0.000 }
gfCNCPoint3[19911] = {X 575.3376, Y 5.0000, Z -4.6667, A 0.000, B 0.000, C 0.000 }
gfCNCPoint3[19912] = {X 575.3372, Y 5.9910, Z -4.6667, A 0.000, B 0.000, C 0.000 }
gfCNCPoint3[19913] = {X 575.2577, Y 6.7687, Z -4.6667, A 0.000, B 0.000, C 0.000 }
gfCNCPoint3[19914] = {X 575.0417, Y 7.5201, Z -4.6667, A 0.000, B 0.000, C 0.000 }
gfCNCPoint3[19915] = {X 574.6962, Y 8.2215, Z -4.6667, A 0.000, B 0.000, C 0.000 }
gfCNCPoint3[19916] = {X 575.2866, Y 9.6569, Z -4.6667, A 0.000, B 0.000, C 0.000 }
gfCNCPoint3[19917] = {X 578.9730, Y 18.7103, Z -4.6667, A 0.000, B 0.000, C 0.000 }
gfCNCPoint3[19918] = {X 580.9325, Y 23.5224, Z -4.6667, A 0.000, B 0.000, C 0.000 }
gfCNCPoint3[19919] = {X 581.1912, Y 24.1578, Z -4.6667, A 0.000, B 0.000, C 0.000 }
gfCNCPoint3[19920] = {X 581.4509, Y 23.5227, Z -4.6667, A 0.000, B 0.000, C 0.000 }
gfCNCPoint3[19921] = {X 587.7570, Y 8.1000, Z -4.6667, A 0.000, B 0.000, C 0.000 }
gfCNCPoint3[19922] = {X 587.4434, Y 7.4143, Z -4.6667, A 0.000, B 0.000, C 0.000 }
gfCNCPoint3[19923] = {X 587.2515, Y 6.6852, Z -4.6667, A 0.000, B 0.000, C 0.000 }
gfCNCPoint3[19924] = {X 587.1870, Y 5.9340, Z -4.6667, A 0.000, B 0.000, C 0.000 }
gfCNCPoint3[19925] = {X 587.1870, Y 5.0000, Z -4.6667, A 0.000, B 0.000, C 0.000 }
gfCNCPoint3[19926] = {X 587.2780, Y 4.1097, Z -4.6667, A 0.000, B 0.000, C 0.000 }
gfCNCPoint3[19927] = {X 587.5473, Y 3.2562, Z -4.6667, A 0.000, B 0.000, C 0.000 }
gfCNCPoint3[19928] = {X 588.0582, Y 2.3717, Z -4.6667, A 0.000, B 0.000, C 0.000 }
gfCNCPoint3[19929] = {X 588.7592, Y 1.6289, Z -4.6667, A 0.000, B 0.000, C 0.000 }
gfCNCPoint3[19930] = {X 589.6127, Y 1.0678, Z -4.6667, A 0.000, B 0.000, C 0.000 }
gfCNCPoint3[19931] = {X 590.5725, Y 0.7185, Z -4.6667, A 0.000, B 0.000, C 0.000 }
gfCNCPoint3[19932] = {X 591.5870, Y 0.6000, Z -4.6667, A 0.000, B 0.000, C 0.000 }
gfCNCPoint3[19933] = {X 600.0000, Y 0.6000, Z -4.6667, A 0.000, B 0.000, C 0.000 }
gfCNCPoint3[19934] = {X 600.8720, Y 0.6873, Z -4.6667, A 0.000, B 0.000, C 0.000 }
gfCNCPoint3[19935] = {X 601.7094, Y 0.9456, Z -4.6667, A 0.000, B 0.000, C 0.000 }
gfCNCPoint3[19936] = {X 602.4790, Y 1.3648, Z -4.6667, A 0.000, B 0.000, C 0.000 }
gfCNCPoint3[19937] = {X 603.1503, Y 1.9282, Z -4.6667, A 0.000, B 0.000, C 0.000 }
gfCNCPoint3[19938] = {X 603.6966, Y 2.6135, Z -4.6667, A 0.000, B 0.000, C 0.000 }
gfCNCPoint3[19939] = {X 603.6966, Y 1.8141, Z -4.6667, A 0.000, B 0.000, C 0.000 }
gfCNCPoint3[19940] = {X 602.9513, Y 1.1136, Z -4.6667, A 0.000, B 0.000, C 0.000 }
gfCNCPoint3[19941] = {X 602.0763, Y 0.5837, Z -4.6667, A 0.000, B 0.000, C 0.000 }
gfCNCPoint3[19942] = {X 601.1101, Y 0.2479, Z -4.6667, A 0.000, B 0.000, C 0.000 }
gfCNCPoint3[19943] = {X 600.0951, Y 0.1209, Z -4.6667, A 0.000, B 0.000, C 0.000 }
gfCNCPoint3[19944] = {X 600.0949, Y -0.0187, Z -4.6667, A 0.000, B 0.000, C 0.000 }
gfCNCPoint3[19945] = {X 600.0672, Y -0.0698, Z -4.6667, A 0.000, B 0.000, C 0.000 }
gfCNCPoint3[19946] = {X 600.0148, Y -0.0950, Z -4.6667, A 0.000, B 0.000, C 0.000 }
gfCNCPoint3[19947] = {X 351.5662, Y -0.0950, Z -4.6667, A 0.000, B 0.000, C 0.000 }
gfCNCPoint3[19948] = {X 351.4056, Y -0.1250, Z -4.6667, A 0.000, B 0.000, C 0.000 }
gfCNCPoint3[19949] = {X 348.9093, Y -0.4714, Z -4.6667, A 0.000, B 0.000, C 0.000 }
gfCNCPoint3[19950] = {X 346.3914, Y -0.5822, Z -4.6667, A 0.000, B 0.000, C 0.000 }
gfCNCPoint3[19951] = {X 343.8743, Y -0.4564, Z -4.6667, A 0.000, B 0.000, C 0.000 }
gfCNCPoint3[19952] = {X 341.3801, Y -0.0950, Z -4.6667, A 0.000, B 0.000, C 0.000 }
gfCNCPoint3[19953] = {X -0.0148, Y -0.0950, Z -4.6667, A 0.000, B 0.000, C 0.000 }
gfCNCPoint3[19954] = {X -0.0672, Y -0.0698, Z -4.6667, A 0.000, B 0.000, C 0.000 }
gfCNCPoint3[19955] = {X -0.0949, Y -0.0187, Z -4.6667, A 0.000, B 0.000, C 0.000 }
gfCNCPoint3[19956] = {X -0.0966, Y 0.8568, Z -4.6667, A 0.000, B 0.000, C 0.000 }
gfCNCPoint3[19957] = {X -0.0966, Y 8.7891, Z -4.6667, A 0.000, B 0.000, C 0.000 }
gfCNCPoint3[19958] = {X -0.7633, Y 8.9979, Z -4.6667, A 0.000, B 0.000, C 0.000 }
gfCNCPoint3[19959] = {X -1.3934, Y 9.2998, Z -4.6667, A 0.000, B 0.000, C 0.000 }
gfCNCPoint3[19960] = {X -1.9904, Y 9.6404, Z -4.6667, A 0.000, B 0.000, C 0.000 }
gfCNCPoint3[19961] = {X -2.6455, Y 10.0884, Z -4.6667, A 0.000, B 0.000, C 0.000 }
gfCNCPoint3[19962] = {X -3.2193, Y 10.6367, Z -4.6667, A 0.000, B 0.000, C 0.000 }
gfCNCPoint3[19963] = {X -3.6966, Y 11.2707, Z -4.6667, A 0.000, B 0.000, C 0.000 }
gfCNCPoint3[19964] = {X -3.6966, Y 12.3463, Z -4.6667, A 0.000, B 0.000, C 0.000 }
gfCNCPoint3[19965] = {X -3.2332, Y 11.4384, Z -4.6667, A 0.000, B 0.000, C 0.000 }
gfCNCPoint3[19966] = {X -2.5734, Y 10.6616, Z -4.6667, A 0.000, B 0.000, C 0.000 }
gfCNCPoint3[19967] = {X -1.7526, Y 10.0573, Z -4.6667, A 0.000, B 0.000, C 0.000 }
gfCNCPoint3[19968] = {X -1.0994, Y 9.6852, Z -4.6667, A 0.000, B 0.000, C 0.000 }
gfCNCPoint3[19969] = {X -0.1608, Y 9.3012, Z -4.6667, A 0.000, B 0.000, C 0.000 }
gfCNCPoint3[19970] = {X 0.8408, Y 9.1423, Z -4.6667, A 0.000, B 0.000, C 0.000 }
gfCNCPoint3[19971] = {X 1.8522, Y 9.2169, Z -4.6667, A 0.000, B 0.000, C 0.000 }
gfCNCPoint3[19972] = {X 2.2349, Y 9.3081, Z -4.6667, A 0.000, B 0.000, C 0.000 }
gfCNCPoint3[19973] = {X 2.6079, Y 9.4331, Z -4.6667, A 0.000, B 0.000, C 0.000 }
gfCNCPoint3[19974] = {X 3.3767, Y 9.0700, Z -4.6667, A 0.000, B 0.000, C 0.000 }
gfCNCPoint3[19975] = {X 4.1713, Y 8.7676, Z -4.6667, A 0.000, B 0.000, C 0.000 }
gfCNCPoint3[19976] = {X 6.0883, Y 8.0972, Z -4.6667, A 0.000, B 0.000, C 0.000 }
gfCNCPoint3[19977] = {X 8.0559, Y 7.5945, Z -4.6667, A 0.000, B 0.000, C 0.000 }
gfCNCPoint3[19978] = {X 10.0595, Y 7.2632, Z -4.6667, A 0.000, B 0.000, C 0.000 }
gfCNCPoint3[19979] = {X 12.0843, Y 7.1059, Z -4.6667, A 0.000, B 0.000, C 0.000 }
gfCNCPoint3[19980] = {X 14.1150, Y 7.1237, Z -4.6667, A 0.000, B 0.000, C 0.000 }
gfCNCPoint3[19981] = {X 16.1367, Y 7.3164, Z -4.6667, A 0.000, B 0.000, C 0.000 }
gfCNCPoint3[19982] = {X 16.5421, Y 7.3732, Z -4.6667, A 0.000, B 0.000, C 0.000 }
gfCNCPoint3[19983] = {X 18.2860, Y 7.7305, Z -4.6667, A 0.000, B 0.000, C 0.000 }
gfCNCPoint3[19984] = {X 19.9847, Y 8.2628, Z -4.6667, A 0.000, B 0.000, C 0.000 }
gfCNCPoint3[19985] = {X 21.6206, Y 8.9646, Z -4.6667, A 0.000, B 0.000, C 0.000 }
gfCNCPoint3[19986] = {X 23.1769, Y 9.8286, Z -4.6667, A 0.000, B 0.000, C 0.000 }
gfCNCPoint3[19987] = {X 24.6376, Y 10.8461, Z -4.6667, A 0.000, B 0.000, C 0.000 }
gfCNCPoint3[19988] = {X 25.7300, Y 11.8014, Z -4.6667, A 0.000, B 0.000, C 0.000 }
gfCNCPoint3[19989] = {X 26.7099, Y 12.8720, Z -4.6667, A 0.000, B 0.000, C 0.000 }
gfCNCPoint3[19990] = {X 27.5651, Y 14.0445, Z -4.6667, A 0.000, B 0.000, C 0.000 }
gfCNCPoint3[19991] = {X 28.2851, Y 15.3045, Z -4.6667, A 0.000, B 0.000, C 0.000 }
gfCNCPoint3[19992] = {X 28.8610, Y 16.6366, Z -4.6667, A 0.000, B 0.000, C 0.000 }
gfCNCPoint3[19993] = {X 29.3381, Y 18.3011, Z -4.6667, A 0.000, B 0.000, C 0.000 }
gfCNCPoint3[19994] = {X 29.6211, Y 20.0093, Z -4.6667, A 0.000, B 0.000, C 0.000 }
gfCNCPoint3[19995] = {X 29.7064, Y 21.7387, Z -4.6667, A 0.000, B 0.000, C 0.000 }
gfCNCPoint3[19996] = {X 29.5926, Y 23.4664, Z -4.6667, A 0.000, B 0.000, C 0.000 }
gfCNCPoint3[19997] = {X 29.2814, Y 25.1697, Z -4.6667, A 0.000, B 0.000, C 0.000 }
gfCNCPoint3[19998] = {X 28.9227, Y 26.3893, Z -4.6667, A 0.000, B 0.000, C 0.000 }
gfCNCPoint3[19999] = {X 28.4345, Y 27.5630, Z -4.6667, A 0.000, B 0.000, C 0.000 }
gfCNCPoint3[20000] = {X 27.8227, Y 28.6772, Z -4.6667, A 0.000, B 0.000, C 0.000 }
gfCNCPoint3[20001] = {X 27.5100, Y 29.1540, Z -4.6667, A 0.000, B 0.000, C 0.000 }
gfCNCPoint3[20002] = {X 27.1746, Y 29.6150, Z -4.6667, A 0.000, B 0.000, C 0.000 }
gfCNCPoint3[20003] = {X 26.3575, Y 30.5722, Z -4.6667, A 0.000, B 0.000, C 0.000 }
gfCNCPoint3[20004] = {X 25.4430, Y 31.4366, Z -4.6667, A 0.000, B 0.000, C 0.000 }
gfCNCPoint3[20005] = {X 25.6936, Y 31.5323, Z -4.6667, A 0.000, B 0.000, C 0.000 }
gfCNCPoint3[20006] = {X 25.9379, Y 31.6430, Z -4.6667, A 0.000, B 0.000, C 0.000 }
gfCNCPoint3[20007] = {X 26.6626, Y 32.0902, Z -4.6667, A 0.000, B 0.000, C 0.000 }
gfCNCPoint3[20008] = {X 27.2876, Y 32.6687, Z -4.6667, A 0.000, B 0.000, C 0.000 }
gfCNCPoint3[20009] = {X 27.6591, Y 33.1493, Z -4.6667, A 0.000, B 0.000, C 0.000 }
gfCNCPoint3[20010] = {X 27.9609, Y 33.6765, Z -4.6667, A 0.000, B 0.000, C 0.000 }
gfCNCPoint3[20011] = {X 30.9820, Y 39.9182, Z -4.6667, A 0.000, B 0.000, C 0.000 }
gfCNCPoint3[20012] = {X 31.3085, Y 40.8441, Z -4.6667, A 0.000, B 0.000, C 0.000 }
gfCNCPoint3[20013] = {X 31.4215, Y 41.8194, Z -4.6667, A 0.000, B 0.000, C 0.000 }
gfCNCPoint3[20014] = {X 31.3155, Y 42.7955, Z -4.6667, A 0.000, B 0.000, C 0.000 }
gfCNCPoint3[20015] = {X 30.9956, Y 43.7238, Z -4.6667, A 0.000, B 0.000, C 0.000 }
gfCNCPoint3[20016] = {X 30.4779, Y 44.5580, Z -4.6667, A 0.000, B 0.000, C 0.000 }
gfCNCPoint3[20017] = {X 29.7880, Y 45.2567, Z -4.6667, A 0.000, B 0.000, C 0.000 }
gfCNCPoint3[20018] = {X 29.2518, Y 45.6902, Z -4.6667, A 0.000, B 0.000, C 0.000 }
gfCNCPoint3[20019] = {X 28.5407, Y 46.1589, Z -4.6667, A 0.000, B 0.000, C 0.000 }
gfCNCPoint3[20020] = {X 27.7529, Y 46.4824, Z -4.6667, A 0.000, B 0.000, C 0.000 }
gfCNCPoint3[20021] = {X 26.9175, Y 46.6485, Z -4.6667, A 0.000, B 0.000, C 0.000 }
gfCNCPoint3[20022] = {X 26.0659, Y 46.6511, Z -4.6667, A 0.000, B 0.000, C 0.000 }
gfCNCPoint3[20023] = {X 25.2295, Y 46.4900, Z -4.6667, A 0.000, B 0.000, C 0.000 }
gfCNCPoint3[20024] = {X 23.4342, Y 47.4357, Z -4.6667, A 0.000, B 0.000, C 0.000 }
gfCNCPoint3[20025] = {X 21.5776, Y 48.2548, Z -4.6667, A 0.000, B 0.000, C 0.000 }
gfCNCPoint3[20026] = {X 19.6687, Y 48.9432, Z -4.6667, A 0.000, B 0.000, C 0.000 }
gfCNCPoint3[20027] = {X 19.5106, Y 48.9961, Z -4.6667, A 0.000, B 0.000, C 0.000 }
gfCNCPoint3[20028] = {X 17.5869, Y 49.5245, Z -4.6667, A 0.000, B 0.000, C 0.000 }
gfCNCPoint3[20029] = {X 15.6245, Y 49.8832, Z -4.6667, A 0.000, B 0.000, C 0.000 }
gfCNCPoint3[20030] = {X 13.6383, Y 50.0695, Z -4.6667, A 0.000, B 0.000, C 0.000 }
gfCNCPoint3[20031] = {X 11.6434, Y 50.0819, Z -4.6667, A 0.000, B 0.000, C 0.000 }
gfCNCPoint3[20032] = {X 9.6551, Y 49.9203, Z -4.6667, A 0.000, B 0.000, C 0.000 }
gfCNCPoint3[20033] = {X 7.6884, Y 49.5859, Z -4.6667, A 0.000, B 0.000, C 0.000 }
gfCNCPoint3[20034] = {X 6.2184, Y 49.2051, Z -4.6667, A 0.000, B 0.000, C 0.000 }
gfCNCPoint3[20035] = {X 4.7888, Y 48.6929, Z -4.6667, A 0.000, B 0.000, C 0.000 }
gfCNCPoint3[20036] = {X 3.4114, Y 48.0535, Z -4.6667, A 0.000, B 0.000, C 0.000 }
gfCNCPoint3[20037] = {X 1.9574, Y 47.2014, Z -4.6667, A 0.000, B 0.000, C 0.000 }
gfCNCPoint3[20038] = {X 0.5963, Y 46.2077, Z -4.6667, A 0.000, B 0.000, C 0.000 }
gfCNCPoint3[20039] = {X -0.4516, Y 45.2752, Z -4.6667, A 0.000, B 0.000, C 0.000 }
gfCNCPoint3[20040] = {X -1.3936, Y 44.2358, Z -4.6667, A 0.000, B 0.000, C 0.000 }
gfCNCPoint3[20041] = {X -2.2190, Y 43.1015, Z -4.6667, A 0.000, B 0.000, C 0.000 }
gfCNCPoint3[20042] = {X -2.9181, Y 41.8854, Z -4.6667, A 0.000, B 0.000, C 0.000 }
gfCNCPoint3[20043] = {X -3.3445, Y 40.9532, Z -4.6667, A 0.000, B 0.000, C 0.000 }
gfCNCPoint3[20044] = {X -3.6966, Y 39.9905, Z -4.6667, A 0.000, B 0.000, C 0.000 }
gfCNCPoint3[20045] = {X -3.6966, Y 41.3539, Z -4.6667, A 0.000, B 0.000, C 0.000 }
gfCNCPoint3[20046] = {X -3.0109, Y 42.7248, Z -4.6667, A 0.000, B 0.000, C 0.000 }
gfCNCPoint3[20047] = {X -2.1749, Y 44.0096, Z -4.6667, A 0.000, B 0.000, C 0.000 }
gfCNCPoint3[20048] = {X -1.1993, Y 45.1919, Z -4.6667, A 0.000, B 0.000, C 0.000 }
gfCNCPoint3[20049] = {X -0.0966, Y 46.2566, Z -4.6667, A 0.000, B 0.000, C 0.000 }
gfCNCPoint3[20050] = {X -0.0966, Y 99.1432, Z -4.6667, A 0.000, B 0.000, C 0.000 }
gfCNCPoint3[20051] = {X -0.0949, Y 100.0187, Z -4.6667, A 0.000, B 0.000, C 0.000 }
gfCNCPoint3[20052] = {X -0.0672, Y 100.0698, Z -4.6667, A 0.000, B 0.000, C 0.000 }
gfCNCPoint3[20053] = {X -0.0148, Y 100.0950, Z -4.6667, A 0.000, B 0.000, C 0.000 }
gfCNCPoint3[20054] = {X 120.5926, Y 100.0950, Z -4.6667, A 0.000, B 0.000, C 0.000 }
gfCNCPoint3[20055] = {X 121.0614, Y 100.8812, Z -4.6667, A 0.000, B 0.000, C 0.000 }
gfCNCPoint3[20056] = {X 121.6687, Y 101.5661, Z -4.6667, A 0.000, B 0.000, C 0.000 }
gfCNCPoint3[20057] = {X 122.3932, Y 102.1254, Z -4.6667, A 0.000, B 0.000, C 0.000 }
gfCNCPoint3[20058] = {X 123.2095, Y 102.5396, Z -4.6667, A 0.000, B 0.000, C 0.000 }
gfCNCPoint3[20059] = {X 124.0887, Y 102.7942, Z -4.6667, A 0.000, B 0.000, C 0.000 }
gfCNCPoint3[20060] = {X 125.0000, Y 102.8800, Z -4.6667, A 0.000, B 0.000, C 0.000 }
gfCNCPoint3[20061] = {X 143.7791, Y 102.8800, Z -4.6667, A 0.000, B 0.000, C 0.000 }
gfCNCPoint3[20062] = {X 144.6904, Y 102.7942, Z -4.6667, A 0.000, B 0.000, C 0.000 }
gfCNCPoint3[20063] = {X 145.5697, Y 102.5396, Z -4.6667, A 0.000, B 0.000, C 0.000 }
gfCNCPoint3[20064] = {X 146.3859, Y 102.1254, Z -4.6667, A 0.000, B 0.000, C 0.000 }
gfCNCPoint3[20065] = {X 147.1104, Y 101.5661, Z -4.6667, A 0.000, B 0.000, C 0.000 }
gfCNCPoint3[20066] = {X 147.7178, Y 100.8812, Z -4.6667, A 0.000, B 0.000, C 0.000 }
gfCNCPoint3[20067] = {X 148.1865, Y 100.0950, Z -4.6667, A 0.000, B 0.000, C 0.000 }
gfCNCPoint3[20068] = {X 150.8377, Y 100.0950, Z -4.6667, A 0.000, B 0.000, C 0.000 }
gfCNCPoint3[20069] = {X 150.8377, Y 95.2950, Z -4.6667, A 0.000, B 0.000, C 0.000 }
gfCNCPoint3[20070] = {X 187.9256, Y 95.2950, Z -4.6667, A 0.000, B 0.000, C 0.000 }
gfCNCPoint3[20071] = {X 187.9777, Y 95.0990, Z -4.6667, A 0.000, B 0.000, C 0.000 }
gfCNCPoint3[20072] = {X 188.0352, Y 94.9045, Z -4.6667, A 0.000, B 0.000, C 0.000 }
gfCNCPoint3[20073] = {X 187.2619, Y 94.0602, Z -4.6667, A 0.000, B 0.000, C 0.000 }
gfCNCPoint3[20074] = {X 151.4055, Y 94.0602, Z -4.6667, A 0.000, B 0.000, C 0.000 }
gfCNCPoint3[20075] = {X 150.7058, Y 94.8354, Z -4.6667, A 0.000, B 0.000, C 0.000 }
gfCNCPoint3[20076] = {X 150.7755, Y 95.0642, Z -4.6667, A 0.000, B 0.000, C 0.000 }
gfCNCPoint3[20077] = {X 150.8377, Y 95.2950, Z -4.6667, A 0.000, B 0.000, C 0.000 }
gfCNCPoint3[20078] = {X 150.8377, Y 97.6950, Z -4.6667, A 0.000, B 0.000, C 0.000 }
gfCNCPoint3[20079] = {X 190.1070, Y 97.6950, Z -4.6667, A 0.000, B 0.000, C 0.000 }
gfCNCPoint3[20080] = {X 190.1070, Y 97.0659, Z -4.6667, A 0.000, B 0.000, C 0.000 }
gfCNCPoint3[20081] = {X 190.1938, Y 96.1495, Z -4.6667, A 0.000, B 0.000, C 0.000 }
gfCNCPoint3[20082] = {X 190.4511, Y 95.2657, Z -4.6667, A 0.000, B 0.000, C 0.000 }
gfCNCPoint3[20083] = {X 190.8699, Y 94.4460, Z -4.6667, A 0.000, B 0.000, C 0.000 }
gfCNCPoint3[20084] = {X 188.3182, Y 91.6602, Z -4.6667, A 0.000, B 0.000, C 0.000 }
gfCNCPoint3[20085] = {X 150.3387, Y 91.6602, Z -4.6667, A 0.000, B 0.000, C 0.000 }
gfCNCPoint3[20086] = {X 147.8638, Y 94.4021, Z -4.6667, A 0.000, B 0.000, C 0.000 }
gfCNCPoint3[20087] = {X 148.2980, Y 95.2326, Z -4.6667, A 0.000, B 0.000, C 0.000 }
gfCNCPoint3[20088] = {X 148.5664, Y 96.1305, Z -4.6667, A 0.000, B 0.000, C 0.000 }
gfCNCPoint3[20089] = {X 148.6591, Y 97.0630, Z -4.6667, A 0.000, B 0.000, C 0.000 }
gfCNCPoint3[20090] = {X 148.6591, Y 97.6950, Z -4.6667, A 0.000, B 0.000, C 0.000 }
gfCNCPoint3[20091] = {X 150.8377, Y 97.6950, Z -4.6667, A 0.000, B 0.000, C 0.000 }
gfCNCPoint3[20092] = {X 150.8377, Y 100.0950, Z -4.6667, A 0.000, B 0.000, C 0.000 }
gfCNCPoint3[20093] = {X 190.5795, Y 100.0950, Z -4.6667, A 0.000, B 0.000, C 0.000 }
gfCNCPoint3[20094] = {X 191.0483, Y 100.8812, Z -4.6667, A 0.000, B 0.000, C 0.000 }
gfCNCPoint3[20095] = {X 191.6556, Y 101.5660, Z -4.6667, A 0.000, B 0.000, C 0.000 }
gfCNCPoint3[20096] = {X 192.3802, Y 102.1254, Z -4.6667, A 0.000, B 0.000, C 0.000 }
gfCNCPoint3[20097] = {X 193.1964, Y 102.5396, Z -4.6667, A 0.000, B 0.000, C 0.000 }
gfCNCPoint3[20098] = {X 194.0757, Y 102.7942, Z -4.6667, A 0.000, B 0.000, C 0.000 }
gfCNCPoint3[20099] = {X 194.9870, Y 102.8800, Z -4.6667, A 0.000, B 0.000, C 0.000 }
gfCNCPoint3[20100] = {X 212.6141, Y 102.8800, Z -4.6667, A 0.000, B 0.000, C 0.000 }
gfCNCPoint3[20101] = {X 213.0066, Y 102.8642, Z -4.6667, A 0.000, B 0.000, C 0.000 }
gfCNCPoint3[20102] = {X 213.3966, Y 102.8169, Z -4.6667, A 0.000, B 0.000, C 0.000 }
gfCNCPoint3[20103] = {X 213.7865, Y 102.8642, Z -4.6667, A 0.000, B 0.000, C 0.000 }
gfCNCPoint3[20104] = {X 214.1790, Y 102.8800, Z -4.6667, A 0.000, B 0.000, C 0.000 }
gfCNCPoint3[20105] = {X 233.4798, Y 102.8800, Z -4.6667, A 0.000, B 0.000, C 0.000 }
gfCNCPoint3[20106] = {X 234.3911, Y 102.7942, Z -4.6667, A 0.000, B 0.000, C 0.000 }
gfCNCPoint3[20107] = {X 235.2703, Y 102.5396, Z -4.6667, A 0.000, B 0.000, C 0.000 }
gfCNCPoint3[20108] = {X 236.0866, Y 102.1254, Z -4.6667, A 0.000, B 0.000, C 0.000 }
gfCNCPoint3[20109] = {X 236.8111, Y 101.5661, Z -4.6667, A 0.000, B 0.000, C 0.000 }
gfCNCPoint3[20110] = {X 237.4184, Y 100.8812, Z -4.6667, A 0.000, B 0.000, C 0.000 }
gfCNCPoint3[20111] = {X 237.8872, Y 100.0950, Z -4.6667, A 0.000, B 0.000, C 0.000 }
gfCNCPoint3[20112] = {X 261.4776, Y 100.0950, Z -4.6667, A 0.000, B 0.000, C 0.000 }
gfCNCPoint3[20113] = {X 261.4776, Y 90.4950, Z -4.6667, A 0.000, B 0.000, C 0.000 }
gfCNCPoint3[20114] = {X 266.0962, Y 90.4950, Z -4.6667, A 0.000, B 0.000, C 0.000 }
gfCNCPoint3[20115] = {X 266.1752, Y 90.3747, Z -4.6667, A 0.000, B 0.000, C 0.000 }
gfCNCPoint3[20116] = {X 266.2556, Y 90.2554, Z -4.6667, A 0.000, B 0.000, C 0.000 }
gfCNCPoint3[20117] = {X 263.5096, Y 89.1789, Z -4.6667, A 0.000, B 0.000, C 0.000 }
gfCNCPoint3[20118] = {X 261.4776, Y 90.4950, Z -4.6667, A 0.000, B 0.000, C 0.000 }
gfCNCPoint3[20119] = {X 261.4776, Y 92.8950, Z -4.6667, A 0.000, B 0.000, C 0.000 }
gfCNCPoint3[20120] = {X 267.4974, Y 92.8950, Z -4.6667, A 0.000, B 0.000, C 0.000 }
gfCNCPoint3[20121] = {X 267.8429, Y 92.2375, Z -4.6667, A 0.000, B 0.000, C 0.000 }
gfCNCPoint3[20122] = {X 268.2378, Y 91.6085, Z -4.6667, A 0.000, B 0.000, C 0.000 }
gfCNCPoint3[20123] = {X 269.1700, Y 90.4463, Z -4.6667, A 0.000, B 0.000, C 0.000 }
gfCNCPoint3[20124] = {X 270.2694, Y 89.4409, Z -4.6667, A 0.000, B 0.000, C 0.000 }
gfCNCPoint3[20125] = {X 270.2694, Y 89.2510, Z -4.6667, A 0.000, B 0.000, C 0.000 }
gfCNCPoint3[20126] = {X 263.2387, Y 86.4949, Z -4.6667, A 0.000, B 0.000, C 0.000 }
gfCNCPoint3[20127] = {X 253.3577, Y 92.8950, Z -4.6667, A 0.000, B 0.000, C 0.000 }
gfCNCPoint3[20128] = {X 261.4776, Y 92.8950, Z -4.6667, A 0.000, B 0.000, C 0.000 }
gfCNCPoint3[20129] = {X 261.4776, Y 95.2950, Z -4.6667, A 0.000, B 0.000, C 0.000 }
gfCNCPoint3[20130] = {X 269.1714, Y 95.2950, Z -4.6667, A 0.000, B 0.000, C 0.000 }
gfCNCPoint3[20131] = {X 269.5515, Y 94.1745, Z -4.6667, A 0.000, B 0.000, C 0.000 }
gfCNCPoint3[20132] = {X 270.1082, Y 93.1303, Z -4.6667, A 0.000, B 0.000, C 0.000 }
gfCNCPoint3[20133] = {X 270.8267, Y 92.1901, Z -4.6667, A 0.000, B 0.000, C 0.000 }
gfCNCPoint3[20134] = {X 271.6880, Y 91.3787, Z -4.6667, A 0.000, B 0.000, C 0.000 }
gfCNCPoint3[20135] = {X 272.6694, Y 90.7176, Z -4.6667, A 0.000, B 0.000, C 0.000 }
gfCNCPoint3[20136] = {X 272.6694, Y 87.6139, Z -4.6667, A 0.000, B 0.000, C 0.000 }
gfCNCPoint3[20137] = {X 262.9678, Y 83.8109, Z -4.6667, A 0.000, B 0.000, C 0.000 }
gfCNCPoint3[20138] = {X 245.2378, Y 95.2950, Z -4.6667, A 0.000, B 0.000, C 0.000 }
gfCNCPoint3[20139] = {X 261.4776, Y 95.2950, Z -4.6667, A 0.000, B 0.000, C 0.000 }
gfCNCPoint3[20140] = {X 261.4776, Y 97.6950, Z -4.6667, A 0.000, B 0.000, C 0.000 }
gfCNCPoint3[20141] = {X 271.3527, Y 97.6950, Z -4.6667, A 0.000, B 0.000, C 0.000 }
gfCNCPoint3[20142] = {X 271.3529, Y 97.0186, Z -4.6667, A 0.000, B 0.000, C 0.000 }
gfCNCPoint3[20143] = {X 271.4810, Y 95.9545, Z -4.6667, A 0.000, B 0.000, C 0.000 }
gfCNCPoint3[20144] = {X 271.8382, Y 94.9440, Z -4.6667, A 0.000, B 0.000, C 0.000 }
gfCNCPoint3[20145] = {X 272.4073, Y 94.0359, Z -4.6667, A 0.000, B 0.000, C 0.000 }
gfCNCPoint3[20146] = {X 273.1610, Y 93.2739, Z -4.6667, A 0.000, B 0.000, C 0.000 }
gfCNCPoint3[20147] = {X 274.0629, Y 92.6949, Z -4.6667, A 0.000, B 0.000, C 0.000 }
gfCNCPoint3[20148] = {X 275.0694, Y 92.3266, Z -4.6667, A 0.000, B 0.000, C 0.000 }
gfCNCPoint3[20149] = {X 275.0694, Y 85.9769, Z -4.6667, A 0.000, B 0.000, C 0.000 }
gfCNCPoint3[20150] = {X 262.6989, Y 81.1277, Z -4.6667, A 0.000, B 0.000, C 0.000 }
gfCNCPoint3[20151] = {X 262.5786, Y 81.2035, Z -4.6667, A 0.000, B 0.000, C 0.000 }
gfCNCPoint3[20152] = {X 238.3587, Y 96.8913, Z -4.6667, A 0.000, B 0.000, C 0.000 }
gfCNCPoint3[20153] = {X 238.3598, Y 97.0659, Z -4.6667, A 0.000, B 0.000, C 0.000 }
gfCNCPoint3[20154] = {X 238.3598, Y 97.6950, Z -4.6667, A 0.000, B 0.000, C 0.000 }
gfCNCPoint3[20155] = {X 261.4776, Y 97.6950, Z -4.6667, A 0.000, B 0.000, C 0.000 }
gfCNCPoint3[20156] = {X 261.4776, Y 100.0950, Z -4.6667, A 0.000, B 0.000, C 0.000 }
gfCNCPoint3[20157] = {X 271.8253, Y 100.0950, Z -4.6667, A 0.000, B 0.000, C 0.000 }
gfCNCPoint3[20158] = {X 272.2940, Y 100.8812, Z -4.6667, A 0.000, B 0.000, C 0.000 }
gfCNCPoint3[20159] = {X 272.9014, Y 101.5661, Z -4.6667, A 0.000, B 0.000, C 0.000 }
gfCNCPoint3[20160] = {X 273.6259, Y 102.1254, Z -4.6667, A 0.000, B 0.000, C 0.000 }
gfCNCPoint3[20161] = {X 274.4421, Y 102.5396, Z -4.6667, A 0.000, B 0.000, C 0.000 }
gfCNCPoint3[20162] = {X 275.3214, Y 102.7942, Z -4.6667, A 0.000, B 0.000, C 0.000 }
gfCNCPoint3[20163] = {X 276.2327, Y 102.8800, Z -4.6667, A 0.000, B 0.000, C 0.000 }
gfCNCPoint3[20164] = {X 292.7731, Y 102.8800, Z -4.6667, A 0.000, B 0.000, C 0.000 }
gfCNCPoint3[20165] = {X 293.6844, Y 102.7942, Z -4.6667, A 0.000, B 0.000, C 0.000 }
gfCNCPoint3[20166] = {X 294.5636, Y 102.5396, Z -4.6667, A 0.000, B 0.000, C 0.000 }
gfCNCPoint3[20167] = {X 295.3799, Y 102.1254, Z -4.6667, A 0.000, B 0.000, C 0.000 }
gfCNCPoint3[20168] = {X 296.1044, Y 101.5661, Z -4.6667, A 0.000, B 0.000, C 0.000 }
gfCNCPoint3[20169] = {X 296.7117, Y 100.8812, Z -4.6667, A 0.000, B 0.000, C 0.000 }
gfCNCPoint3[20170] = {X 297.1805, Y 100.0950, Z -4.6667, A 0.000, B 0.000, C 0.000 }
gfCNCPoint3[20171] = {X 319.1327, Y 100.0950, Z -4.6667, A 0.000, B 0.000, C 0.000 }
gfCNCPoint3[20172] = {X 321.4361, Y 100.8685, Z -4.6667, A 0.000, B 0.000, C 0.000 }
gfCNCPoint3[20173] = {X 323.7823, Y 101.5005, Z -4.6667, A 0.000, B 0.000, C 0.000 }
gfCNCPoint3[20174] = {X 326.1627, Y 101.9887, Z -4.6667, A 0.000, B 0.000, C 0.000 }
gfCNCPoint3[20175] = {X 330.1025, Y 102.5981, Z -4.6667, A 0.000, B 0.000, C 0.000 }
gfCNCPoint3[20176] = {X 334.0644, Y 103.0425, Z -4.6667, A 0.000, B 0.000, C 0.000 }
gfCNCPoint3[20177] = {X 338.0414, Y 103.3211, Z -4.6667, A 0.000, B 0.000, C 0.000 }
gfCNCPoint3[20178] = {X 343.7798, Y 103.5417, Z -4.6667, A 0.000, B 0.000, C 0.000 }
gfCNCPoint3[20179] = {X 349.5223, Y 103.5868, Z -4.6667, A 0.000, B 0.000, C 0.000 }
gfCNCPoint3[20180] = {X 355.2635, Y 103.4563, Z -4.6667, A 0.000, B 0.000, C 0.000 }
gfCNCPoint3[20181] = {X 360.9980, Y 103.1505, Z -4.6667, A 0.000, B 0.000, C 0.000 }
gfCNCPoint3[20182] = {X 364.9921, Y 102.7828, Z -4.6667, A 0.000, B 0.000, C 0.000 }
gfCNCPoint3[20183] = {X 368.9631, Y 102.2185, Z -4.6667, A 0.000, B 0.000, C 0.000 }
gfCNCPoint3[20184] = {X 372.9015, Y 101.4590, Z -4.6667, A 0.000, B 0.000, C 0.000 }
gfCNCPoint3[20185] = {X 375.2305, Y 100.8567, Z -4.6667, A 0.000, B 0.000, C 0.000 }
gfCNCPoint3[20186] = {X 377.5122, Y 100.0950, Z -4.6667, A 0.000, B 0.000, C 0.000 }
gfCNCPoint3[20187] = {X 391.9985, Y 100.0950, Z -4.6667, A 0.000, B 0.000, C 0.000 }
gfCNCPoint3[20188] = {X 392.4673, Y 100.8812, Z -4.6667, A 0.000, B 0.000, C 0.000 }
gfCNCPoint3[20189] = {X 393.0746, Y 101.5661, Z -4.6667, A 0.000, B 0.000, C 0.000 }
gfCNCPoint3[20190] = {X 393.7992, Y 102.1254, Z -4.6667, A 0.000, B 0.000, C 0.000 }
gfCNCPoint3[20191] = {X 394.6154, Y 102.5396, Z -4.6667, A 0.000, B 0.000, C 0.000 }
gfCNCPoint3[20192] = {X 395.4946, Y 102.7942, Z -4.6667, A 0.000, B 0.000, C 0.000 }
gfCNCPoint3[20193] = {X 396.4059, Y 102.8800, Z -4.6667, A 0.000, B 0.000, C 0.000 }
gfCNCPoint3[20194] = {X 415.7067, Y 102.8800, Z -4.6667, A 0.000, B 0.000, C 0.000 }
gfCNCPoint3[20195] = {X 416.6180, Y 102.7942, Z -4.6667, A 0.000, B 0.000, C 0.000 }
gfCNCPoint3[20196] = {X 417.4972, Y 102.5396, Z -4.6667, A 0.000, B 0.000, C 0.000 }
gfCNCPoint3[20197] = {X 418.3135, Y 102.1254, Z -4.6667, A 0.000, B 0.000, C 0.000 }
gfCNCPoint3[20198] = {X 419.0380, Y 101.5661, Z -4.6667, A 0.000, B 0.000, C 0.000 }
gfCNCPoint3[20199] = {X 419.6453, Y 100.8812, Z -4.6667, A 0.000, B 0.000, C 0.000 }
gfCNCPoint3[20200] = {X 420.1141, Y 100.0950, Z -4.6667, A 0.000, B 0.000, C 0.000 }
gfCNCPoint3[20201] = {X 443.7028, Y 100.0950, Z -4.6667, A 0.000, B 0.000, C 0.000 }
gfCNCPoint3[20202] = {X 443.7028, Y 90.4950, Z -4.6667, A 0.000, B 0.000, C 0.000 }
gfCNCPoint3[20203] = {X 448.3231, Y 90.4950, Z -4.6667, A 0.000, B 0.000, C 0.000 }
gfCNCPoint3[20204] = {X 448.4021, Y 90.3747, Z -4.6667, A 0.000, B 0.000, C 0.000 }
gfCNCPoint3[20205] = {X 448.4825, Y 90.2554, Z -4.6667, A 0.000, B 0.000, C 0.000 }
gfCNCPoint3[20206] = {X 445.7353, Y 89.1784, Z -4.6667, A 0.000, B 0.000, C 0.000 }
gfCNCPoint3[20207] = {X 443.7028, Y 90.4950, Z -4.6667, A 0.000, B 0.000, C 0.000 }
gfCNCPoint3[20208] = {X 443.7028, Y 92.8950, Z -4.6667, A 0.000, B 0.000, C 0.000 }
gfCNCPoint3[20209] = {X 449.7243, Y 92.8950, Z -4.6667, A 0.000, B 0.000, C 0.000 }
gfCNCPoint3[20210] = {X 450.0698, Y 92.2375, Z -4.6667, A 0.000, B 0.000, C 0.000 }
gfCNCPoint3[20211] = {X 450.4647, Y 91.6084, Z -4.6667, A 0.000, B 0.000, C 0.000 }
gfCNCPoint3[20212] = {X 451.3969, Y 90.4463, Z -4.6667, A 0.000, B 0.000, C 0.000 }
gfCNCPoint3[20213] = {X 452.4963, Y 89.4409, Z -4.6667, A 0.000, B 0.000, C 0.000 }
gfCNCPoint3[20214] = {X 452.4963, Y 89.2510, Z -4.6667, A 0.000, B 0.000, C 0.000 }
gfCNCPoint3[20215] = {X 445.4643, Y 86.4944, Z -4.6667, A 0.000, B 0.000, C 0.000 }
gfCNCPoint3[20216] = {X 435.5835, Y 92.8950, Z -4.6667, A 0.000, B 0.000, C 0.000 }
gfCNCPoint3[20217] = {X 443.7028, Y 92.8950, Z -4.6667, A 0.000, B 0.000, C 0.000 }
gfCNCPoint3[20218] = {X 443.7028, Y 95.2950, Z -4.6667, A 0.000, B 0.000, C 0.000 }
gfCNCPoint3[20219] = {X 451.3983, Y 95.2950, Z -4.6667, A 0.000, B 0.000, C 0.000 }
gfCNCPoint3[20220] = {X 451.7785, Y 94.1745, Z -4.6667, A 0.000, B 0.000, C 0.000 }
gfCNCPoint3[20221] = {X 452.3351, Y 93.1303, Z -4.6667, A 0.000, B 0.000, C 0.000 }
gfCNCPoint3[20222] = {X 453.0536, Y 92.1901, Z -4.6667, A 0.000, B 0.000, C 0.000 }
gfCNCPoint3[20223] = {X 453.9149, Y 91.3787, Z -4.6667, A 0.000, B 0.000, C 0.000 }
gfCNCPoint3[20224] = {X 454.8963, Y 90.7176, Z -4.6667, A 0.000, B 0.000, C 0.000 }
gfCNCPoint3[20225] = {X 454.8963, Y 87.6139, Z -4.6667, A 0.000, B 0.000, C 0.000 }
gfCNCPoint3[20226] = {X 445.1933, Y 83.8104, Z -4.6667, A 0.000, B 0.000, C 0.000 }
gfCNCPoint3[20227] = {X 427.4642, Y 95.2950, Z -4.6667, A 0.000, B 0.000, C 0.000 }
gfCNCPoint3[20228] = {X 443.7028, Y 95.2950, Z -4.6667, A 0.000, B 0.000, C 0.000 }
gfCNCPoint3[20229] = {X 443.7028, Y 97.6950, Z -4.6667, A 0.000, B 0.000, C 0.000 }
gfCNCPoint3[20230] = {X 453.5796, Y 97.6950, Z -4.6667, A 0.000, B 0.000, C 0.000 }
gfCNCPoint3[20231] = {X 453.5796, Y 97.0659, Z -4.6667, A 0.000, B 0.000, C 0.000 }
gfCNCPoint3[20232] = {X 453.6990, Y 95.9930, Z -4.6667, A 0.000, B 0.000, C 0.000 }
gfCNCPoint3[20233] = {X 454.0514, Y 94.9725, Z -4.6667, A 0.000, B 0.000, C 0.000 }
gfCNCPoint3[20234] = {X 454.6196, Y 94.0545, Z -4.6667, A 0.000, B 0.000, C 0.000 }
gfCNCPoint3[20235] = {X 455.3757, Y 93.2839, Z -4.6667, A 0.000, B 0.000, C 0.000 }
gfCNCPoint3[20236] = {X 456.2827, Y 92.6984, Z -4.6667, A 0.000, B 0.000, C 0.000 }
gfCNCPoint3[20237] = {X 457.2963, Y 92.3266, Z -4.6667, A 0.000, B 0.000, C 0.000 }
gfCNCPoint3[20238] = {X 457.2963, Y 85.9769, Z -4.6667, A 0.000, B 0.000, C 0.000 }
gfCNCPoint3[20239] = {X 444.9224, Y 81.1263, Z -4.6667, A 0.000, B 0.000, C 0.000 }
gfCNCPoint3[20240] = {X 420.5855, Y 96.8914, Z -4.6667, A 0.000, B 0.000, C 0.000 }
gfCNCPoint3[20241] = {X 420.5867, Y 97.0659, Z -4.6667, A 0.000, B 0.000, C 0.000 }
gfCNCPoint3[20242] = {X 420.5867, Y 97.6950, Z -4.6667, A 0.000, B 0.000, C 0.000 }
gfCNCPoint3[20243] = {X 443.7028, Y 97.6950, Z -4.6667, A 0.000, B 0.000, C 0.000 }
gfCNCPoint3[20244] = {X 443.7028, Y 100.0950, Z -4.6667, A 0.000, B 0.000, C 0.000 }
gfCNCPoint3[20245] = {X 454.0522, Y 100.0950, Z -4.6667, A 0.000, B 0.000, C 0.000 }
gfCNCPoint3[20246] = {X 454.5210, Y 100.8812, Z -4.6667, A 0.000, B 0.000, C 0.000 }
gfCNCPoint3[20247] = {X 455.1283, Y 101.5661, Z -4.6667, A 0.000, B 0.000, C 0.000 }
gfCNCPoint3[20248] = {X 455.8528, Y 102.1254, Z -4.6667, A 0.000, B 0.000, C 0.000 }
gfCNCPoint3[20249] = {X 456.6691, Y 102.5396, Z -4.6667, A 0.000, B 0.000, C 0.000 }
gfCNCPoint3[20250] = {X 457.5483, Y 102.7942, Z -4.6667, A 0.000, B 0.000, C 0.000 }
gfCNCPoint3[20251] = {X 458.4596, Y 102.8800, Z -4.6667, A 0.000, B 0.000, C 0.000 }
gfCNCPoint3[20252] = {X 475.0000, Y 102.8800, Z -4.6667, A 0.000, B 0.000, C 0.000 }
gfCNCPoint3[20253] = {X 475.9113, Y 102.7942, Z -4.6667, A 0.000, B 0.000, C 0.000 }
gfCNCPoint3[20254] = {X 476.7905, Y 102.5396, Z -4.6667, A 0.000, B 0.000, C 0.000 }
gfCNCPoint3[20255] = {X 477.6068, Y 102.1254, Z -4.6667, A 0.000, B 0.000, C 0.000 }
gfCNCPoint3[20256] = {X 478.3313, Y 101.5661, Z -4.6667, A 0.000, B 0.000, C 0.000 }
gfCNCPoint3[20257] = {X 478.9386, Y 100.8812, Z -4.6667, A 0.000, B 0.000, C 0.000 }
gfCNCPoint3[20258] = {X 479.4074, Y 100.0950, Z -4.6667, A 0.000, B 0.000, C 0.000 }
gfCNCPoint3[20259] = {X 507.6815, Y 100.0950, Z -4.6667, A 0.000, B 0.000, C 0.000 }
gfCNCPoint3[20260] = {X 507.6815, Y 107.6950, Z -4.6667, A 0.000, B 0.000, C 0.000 }
gfCNCPoint3[20261] = {X 507.6815, Y 107.6950, Z -1.6667, A 0.000, B 0.000, C 0.000 }
gfCNCPoint3[20262] = {X 507.6815, Y 107.6950, Z 11.0000, A 0.000, B 0.000, C 0.000 }
gfCNCPoint3[20263] = {X 108.5564, Y 40.8989, Z 11.0000, A 0.000, B 0.000, C 0.000 }
gfCNCPoint3[20264] = {X 108.5564, Y 40.8989, Z -0.8333, A 0.000, B 0.000, C 0.000 }
gfCNCPoint3[20265] = {X 108.5564, Y 40.8989, Z -4.6667, A 0.000, B 0.000, C 0.000 }
gfCNCPoint3[20266] = {X 108.0669, Y 42.0951, Z -4.6667, A 0.000, B 0.000, C 0.000 }
gfCNCPoint3[20267] = {X 108.0931, Y 42.0495, Z -4.6667, A 0.000, B 0.000, C 0.000 }
gfCNCPoint3[20268] = {X 108.1198, Y 42.0043, Z -4.6667, A 0.000, B 0.000, C 0.000 }
gfCNCPoint3[20269] = {X 108.5454, Y 41.3869, Z -4.6667, A 0.000, B 0.000, C 0.000 }
gfCNCPoint3[20270] = {X 109.0459, Y 40.8286, Z -4.6667, A 0.000, B 0.000, C 0.000 }
gfCNCPoint3[20271] = {X 109.0458, Y 39.7028, Z -4.6667, A 0.000, B 0.000, C 0.000 }
gfCNCPoint3[20272] = {X 108.5564, Y 40.8989, Z -4.6667, A 0.000, B 0.000, C 0.000 }
gfCNCPoint3[20273] = {X 108.5564, Y 40.8989, Z -1.6667, A 0.000, B 0.000, C 0.000 }
gfCNCPoint3[20274] = {X 108.5564, Y 40.8989, Z 11.0000, A 0.000, B 0.000, C 0.000 }
gfCNCPoint3[20275] = {X 95.6832, Y 40.8736, Z 11.0000, A 0.000, B 0.000, C 0.000 }
gfCNCPoint3[20276] = {X 95.6832, Y 40.8736, Z -0.8333, A 0.000, B 0.000, C 0.000 }
gfCNCPoint3[20277] = {X 95.6832, Y 40.8736, Z -4.6667, A 0.000, B 0.000, C 0.000 }
gfCNCPoint3[20278] = {X 95.2111, Y 39.7188, Z -4.6667, A 0.000, B 0.000, C 0.000 }
gfCNCPoint3[20279] = {X 95.2111, Y 40.8686, Z -4.6667, A 0.000, B 0.000, C 0.000 }
gfCNCPoint3[20280] = {X 95.7320, Y 41.4089, Z -4.6667, A 0.000, B 0.000, C 0.000 }
gfCNCPoint3[20281] = {X 96.1554, Y 42.0284, Z -4.6667, A 0.000, B 0.000, C 0.000 }
gfCNCPoint3[20282] = {X 95.6832, Y 40.8736, Z -4.6667, A 0.000, B 0.000, C 0.000 }
gfCNCPoint3[20283] = {X 95.6832, Y 40.8736, Z -1.6667, A 0.000, B 0.000, C 0.000 }
gfCNCPoint3[20284] = {X 95.6832, Y 40.8736, Z 11.0000, A 0.000, B 0.000, C 0.000 }
gfCNCPoint3[20285] = {X -7.6966, Y 43.2956, Z 11.0000, A 0.000, B 0.000, C 0.000 }
gfCNCPoint3[20286] = {X -7.6966, Y 43.2956, Z -1.6667, A 0.000, B 0.000, C 0.000 }
gfCNCPoint3[20287] = {X -7.6966, Y 43.2956, Z -4.6667, A 0.000, B 0.000, C 0.000 }
gfCNCPoint3[20288] = {X -3.6966, Y 30.8016, Z -4.6667, A 0.000, B 0.000, C 0.000 }
gfCNCPoint3[20289] = {X -3.5206, Y 30.2849, Z -4.6667, A 0.000, B 0.000, C 0.000 }
gfCNCPoint3[20290] = {X -3.3259, Y 29.7749, Z -4.6667, A 0.000, B 0.000, C 0.000 }
gfCNCPoint3[20291] = {X -2.7029, Y 28.4549, Z -4.6667, A 0.000, B 0.000, C 0.000 }
gfCNCPoint3[20292] = {X -1.9091, Y 27.2298, Z -4.6667, A 0.000, B 0.000, C 0.000 }
gfCNCPoint3[20293] = {X -0.9589, Y 26.1218, Z -4.6667, A 0.000, B 0.000, C 0.000 }
gfCNCPoint3[20294] = {X 0.1309, Y 25.1506, Z -4.6667, A 0.000, B 0.000, C 0.000 }
gfCNCPoint3[20295] = {X 1.3406, Y 24.3337, Z -4.6667, A 0.000, B 0.000, C 0.000 }
gfCNCPoint3[20296] = {X 0.5800, Y 23.9234, Z -4.6667, A 0.000, B 0.000, C 0.000 }
gfCNCPoint3[20297] = {X -0.0857, Y 23.3724, Z -4.6667, A 0.000, B 0.000, C 0.000 }
gfCNCPoint3[20298] = {X -0.6309, Y 22.7020, Z -4.6667, A 0.000, B 0.000, C 0.000 }
gfCNCPoint3[20299] = {X -1.0345, Y 21.9378, Z -4.6667, A 0.000, B 0.000, C 0.000 }
gfCNCPoint3[20300] = {X -3.6458, Y 15.5423, Z -4.6667, A 0.000, B 0.000, C 0.000 }
gfCNCPoint3[20301] = {X -3.6717, Y 15.4773, Z -4.6667, A 0.000, B 0.000, C 0.000 }
gfCNCPoint3[20302] = {X -3.6966, Y 15.4120, Z -4.6667, A 0.000, B 0.000, C 0.000 }
gfCNCPoint3[20303] = {X -7.6966, Y 4.6495, Z -4.6667, A 0.000, B 0.000, C 0.000 }
gfCNCPoint3[20304] = {X -7.6966, Y 4.6495, Z -1.6667, A 0.000, B 0.000, C 0.000 }
gfCNCPoint3[20305] = {X -7.6966, Y 4.6495, Z 11.0000, A 0.000, B 0.000, C 0.000 }
gfCNCPoint3[20306] = {X -7.6966, Y 16.4126, Z 11.0000, A 0.000, B 0.000, C 0.000 }
gfCNCPoint3[20307] = {X -7.6966, Y 16.4126, Z -1.6667, A 0.000, B 0.000, C 0.000 }
gfCNCPoint3[20308] = {X -7.6966, Y 16.4126, Z -4.6667, A 0.000, B 0.000, C 0.000 }
gfCNCPoint3[20309] = {X -4.8867, Y 16.4126, Z -4.6667, A 0.000, B 0.000, C 0.000 }
gfCNCPoint3[20310] = {X -3.6966, Y 12.5938, Z -4.6667, A 0.000, B 0.000, C 0.000 }
gfCNCPoint3[20311] = {X -3.6606, Y 12.4835, Z -4.6667, A 0.000, B 0.000, C 0.000 }
gfCNCPoint3[20312] = {X -3.6216, Y 12.3741, Z -4.6667, A 0.000, B 0.000, C 0.000 }
gfCNCPoint3[20313] = {X -3.1667, Y 11.4828, Z -4.6667, A 0.000, B 0.000, C 0.000 }
gfCNCPoint3[20314] = {X -2.5189, Y 10.7201, Z -4.6667, A 0.000, B 0.000, C 0.000 }
gfCNCPoint3[20315] = {X -1.7129, Y 10.1268, Z -4.6667, A 0.000, B 0.000, C 0.000 }
gfCNCPoint3[20316] = {X -1.1157, Y 9.7861, Z -4.6667, A 0.000, B 0.000, C 0.000 }
gfCNCPoint3[20317] = {X -0.2299, Y 9.4047, Z -4.6667, A 0.000, B 0.000, C 0.000 }
gfCNCPoint3[20318] = {X 0.7184, Y 9.2294, Z -4.6667, A 0.000, B 0.000, C 0.000 }
gfCNCPoint3[20319] = {X 1.6819, Y 9.2687, Z -4.6667, A 0.000, B 0.000, C 0.000 }
gfCNCPoint3[20320] = {X 2.6127, Y 9.5208, Z -4.6667, A 0.000, B 0.000, C 0.000 }
gfCNCPoint3[20321] = {X 3.3883, Y 9.1521, Z -4.6667, A 0.000, B 0.000, C 0.000 }
gfCNCPoint3[20322] = {X 4.1906, Y 8.8455, Z -4.6667, A 0.000, B 0.000, C 0.000 }
gfCNCPoint3[20323] = {X 6.1023, Y 8.1761, Z -4.6667, A 0.000, B 0.000, C 0.000 }
gfCNCPoint3[20324] = {X 8.0647, Y 7.6740, Z -4.6667, A 0.000, B 0.000, C 0.000 }
gfCNCPoint3[20325] = {X 10.0631, Y 7.3431, Z -4.6667, A 0.000, B 0.000, C 0.000 }
gfCNCPoint3[20326] = {X 12.0825, Y 7.1858, Z -4.6667, A 0.000, B 0.000, C 0.000 }
gfCNCPoint3[20327] = {X 14.1080, Y 7.2033, Z -4.6667, A 0.000, B 0.000, C 0.000 }
gfCNCPoint3[20328] = {X 16.1245, Y 7.3955, Z -4.6667, A 0.000, B 0.000, C 0.000 }
gfCNCPoint3[20329] = {X 17.9477, Y 7.7290, Z -4.6667, A 0.000, B 0.000, C 0.000 }
gfCNCPoint3[20330] = {X 19.7252, Y 8.2540, Z -4.6667, A 0.000, B 0.000, C 0.000 }
gfCNCPoint3[20331] = {X 21.4370, Y 8.9646, Z -4.6667, A 0.000, B 0.000, C 0.000 }
gfCNCPoint3[20332] = {X 23.0639, Y 9.8527, Z -4.6667, A 0.000, B 0.000, C 0.000 }
gfCNCPoint3[20333] = {X 24.5873, Y 10.9083, Z -4.6667, A 0.000, B 0.000, C 0.000 }
gfCNCPoint3[20334] = {X 25.6726, Y 11.8572, Z -4.6667, A 0.000, B 0.000, C 0.000 }
gfCNCPoint3[20335] = {X 26.6462, Y 12.9204, Z -4.6667, A 0.000, B 0.000, C 0.000 }
gfCNCPoint3[20336] = {X 27.4960, Y 14.0849, Z -4.6667, A 0.000, B 0.000, C 0.000 }
gfCNCPoint3[20337] = {X 28.2116, Y 15.3363, Z -4.6667, A 0.000, B 0.000, C 0.000 }
gfCNCPoint3[20338] = {X 28.7842, Y 16.6593, Z -4.6667, A 0.000, B 0.000, C 0.000 }
gfCNCPoint3[20339] = {X 29.2594, Y 18.3157, Z -4.6667, A 0.000, B 0.000, C 0.000 }
gfCNCPoint3[20340] = {X 29.5414, Y 20.0156, Z -4.6667, A 0.000, B 0.000, C 0.000 }
gfCNCPoint3[20341] = {X 29.6264, Y 21.7367, Z -4.6667, A 0.000, B 0.000, C 0.000 }
gfCNCPoint3[20342] = {X 29.5133, Y 23.4561, Z -4.6667, A 0.000, B 0.000, C 0.000 }
gfCNCPoint3[20343] = {X 29.2036, Y 25.1512, Z -4.6667, A 0.000, B 0.000, C 0.000 }
gfCNCPoint3[20344] = {X 28.7614, Y 26.5974, Z -4.6667, A 0.000, B 0.000, C 0.000 }
gfCNCPoint3[20345] = {X 28.1361, Y 27.9743, Z -4.6667, A 0.000, B 0.000, C 0.000 }
gfCNCPoint3[20346] = {X 27.3384, Y 29.2590, Z -4.6667, A 0.000, B 0.000, C 0.000 }
gfCNCPoint3[20347] = {X 26.3814, Y 30.4300, Z -4.6667, A 0.000, B 0.000, C 0.000 }
gfCNCPoint3[20348] = {X 25.2814, Y 31.4677, Z -4.6667, A 0.000, B 0.000, C 0.000 }
gfCNCPoint3[20349] = {X 26.0853, Y 31.8099, Z -4.6667, A 0.000, B 0.000, C 0.000 }
gfCNCPoint3[20350] = {X 26.8040, Y 32.3068, Z -4.6667, A 0.000, B 0.000, C 0.000 }
gfCNCPoint3[20351] = {X 27.4080, Y 32.9381, Z -4.6667, A 0.000, B 0.000, C 0.000 }
gfCNCPoint3[20352] = {X 27.8726, Y 33.6781, Z -4.6667, A 0.000, B 0.000, C 0.000 }
gfCNCPoint3[20353] = {X 30.9100, Y 39.9530, Z -4.6667, A 0.000, B 0.000, C 0.000 }
gfCNCPoint3[20354] = {X 31.2306, Y 40.8622, Z -4.6667, A 0.000, B 0.000, C 0.000 }
gfCNCPoint3[20355] = {X 31.3415, Y 41.8197, Z -4.6667, A 0.000, B 0.000, C 0.000 }
gfCNCPoint3[20356] = {X 31.2374, Y 42.7781, Z -4.6667, A 0.000, B 0.000, C 0.000 }
gfCNCPoint3[20357] = {X 30.9234, Y 43.6895, Z -4.6667, A 0.000, B 0.000, C 0.000 }
gfCNCPoint3[20358] = {X 30.4150, Y 44.5085, Z -4.6667, A 0.000, B 0.000, C 0.000 }
gfCNCPoint3[20359] = {X 29.7377, Y 45.1945, Z -4.6667, A 0.000, B 0.000, C 0.000 }
gfCNCPoint3[20360] = {X 29.2016, Y 45.6280, Z -4.6667, A 0.000, B 0.000, C 0.000 }
gfCNCPoint3[20361] = {X 28.4973, Y 46.0914, Z -4.6667, A 0.000, B 0.000, C 0.000 }
gfCNCPoint3[20362] = {X 27.7167, Y 46.4097, Z -4.6667, A 0.000, B 0.000, C 0.000 }
gfCNCPoint3[20363] = {X 26.8893, Y 46.5709, Z -4.6667, A 0.000, B 0.000, C 0.000 }
gfCNCPoint3[20364] = {X 26.0462, Y 46.5688, Z -4.6667, A 0.000, B 0.000, C 0.000 }
gfCNCPoint3[20365] = {X 25.2196, Y 46.4035, Z -4.6667, A 0.000, B 0.000, C 0.000 }
gfCNCPoint3[20366] = {X 23.4198, Y 47.3539, Z -4.6667, A 0.000, B 0.000, C 0.000 }
gfCNCPoint3[20367] = {X 21.5581, Y 48.1764, Z -4.6667, A 0.000, B 0.000, C 0.000 }
gfCNCPoint3[20368] = {X 19.6436, Y 48.8672, Z -4.6667, A 0.000, B 0.000, C 0.000 }
gfCNCPoint3[20369] = {X 17.7038, Y 49.4143, Z -4.6667, A 0.000, B 0.000, C 0.000 }
gfCNCPoint3[20370] = {X 15.7232, Y 49.7877, Z -4.6667, A 0.000, B 0.000, C 0.000 }
gfCNCPoint3[20371] = {X 13.7174, Y 49.9847, Z -4.6667, A 0.000, B 0.000, C 0.000 }
gfCNCPoint3[20372] = {X 11.7020, Y 50.0035, Z -4.6667, A 0.000, B 0.000, C 0.000 }
gfCNCPoint3[20373] = {X 9.6929, Y 49.8441, Z -4.6667, A 0.000, B 0.000, C 0.000 }
gfCNCPoint3[20374] = {X 7.7057, Y 49.5078, Z -4.6667, A 0.000, B 0.000, C 0.000 }
gfCNCPoint3[20375] = {X 5.8037, Y 48.9870, Z -4.6667, A 0.000, B 0.000, C 0.000 }
gfCNCPoint3[20376] = {X 3.9764, Y 48.2456, Z -4.6667, A 0.000, B 0.000, C 0.000 }
gfCNCPoint3[20377] = {X 2.2493, Y 47.2940, Z -4.6667, A 0.000, B 0.000, C 0.000 }
gfCNCPoint3[20378] = {X 0.6464, Y 46.1453, Z -4.6667, A 0.000, B 0.000, C 0.000 }
gfCNCPoint3[20379] = {X -0.4861, Y 45.1275, Z -4.6667, A 0.000, B 0.000, C 0.000 }
gfCNCPoint3[20380] = {X -1.4918, Y 43.9842, Z -4.6667, A 0.000, B 0.000, C 0.000 }
gfCNCPoint3[20381] = {X -2.3570, Y 42.7312, Z -4.6667, A 0.000, B 0.000, C 0.000 }
gfCNCPoint3[20382] = {X -3.0698, Y 41.3856, Z -4.6667, A 0.000, B 0.000, C 0.000 }
gfCNCPoint3[20383] = {X -3.6204, Y 39.9660, Z -4.6667, A 0.000, B 0.000, C 0.000 }
gfCNCPoint3[20384] = {X -3.6591, Y 39.8437, Z -4.6667, A 0.000, B 0.000, C 0.000 }
gfCNCPoint3[20385] = {X -3.6966, Y 39.7211, Z -4.6667, A 0.000, B 0.000, C 0.000 }
gfCNCPoint3[20386] = {X -4.8469, Y 35.8901, Z -4.6667, A 0.000, B 0.000, C 0.000 }
gfCNCPoint3[20387] = {X -7.9942, Y 36.0023, Z -4.6667, A 0.000, B 0.000, C 0.000 }
gfCNCPoint3[20388] = {X -7.9942, Y 36.0023, Z -1.6667, A 0.000, B 0.000, C 0.000 }
gfCNCPoint3[20389] = {X -7.9942, Y 36.0023, Z 11.0000, A 0.000, B 0.000, C 0.000 }
gfCNCPoint3[20390] = {X 608.0000, Y 40.1197, Z 11.0000, A 0.000, B 0.000, C 0.000 }
gfCNCPoint3[20391] = {X 608.0000, Y 40.1197, Z -1.6667, A 0.000, B 0.000, C 0.000 }
gfCNCPoint3[20392] = {X 608.0000, Y 40.1197, Z -4.6667, A 0.000, B 0.000, C 0.000 }
gfCNCPoint3[20393] = {X 603.6966, Y 47.2356, Z -4.6667, A 0.000, B 0.000, C 0.000 }
gfCNCPoint3[20394] = {X 603.6634, Y 47.2896, Z -4.6667, A 0.000, B 0.000, C 0.000 }
gfCNCPoint3[20395] = {X 603.6294, Y 47.3431, Z -4.6667, A 0.000, B 0.000, C 0.000 }
gfCNCPoint3[20396] = {X 603.0930, Y 48.0159, Z -4.6667, A 0.000, B 0.000, C 0.000 }
gfCNCPoint3[20397] = {X 602.4340, Y 48.5691, Z -4.6667, A 0.000, B 0.000, C 0.000 }
gfCNCPoint3[20398] = {X 601.6783, Y 48.9806, Z -4.6667, A 0.000, B 0.000, C 0.000 }
gfCNCPoint3[20399] = {X 600.8562, Y 49.2343, Z -4.6667, A 0.000, B 0.000, C 0.000 }
gfCNCPoint3[20400] = {X 600.0000, Y 49.3200, Z -4.6667, A 0.000, B 0.000, C 0.000 }
gfCNCPoint3[20401] = {X 593.5565, Y 49.3200, Z -4.6667, A 0.000, B 0.000, C 0.000 }
gfCNCPoint3[20402] = {X 592.5952, Y 49.2117, Z -4.6667, A 0.000, B 0.000, C 0.000 }
gfCNCPoint3[20403] = {X 591.6822, Y 48.8922, Z -4.6667, A 0.000, B 0.000, C 0.000 }
gfCNCPoint3[20404] = {X 590.8631, Y 48.3775, Z -4.6667, A 0.000, B 0.000, C 0.000 }
gfCNCPoint3[20405] = {X 590.1790, Y 47.6935, Z -4.6667, A 0.000, B 0.000, C 0.000 }
gfCNCPoint3[20406] = {X 589.6643, Y 46.8744, Z -4.6667, A 0.000, B 0.000, C 0.000 }
gfCNCPoint3[20407] = {X 589.3448, Y 45.9613, Z -4.6667, A 0.000, B 0.000, C 0.000 }
gfCNCPoint3[20408] = {X 589.2365, Y 45.0000, Z -4.6667, A 0.000, B 0.000, C 0.000 }
gfCNCPoint3[20409] = {X 589.2365, Y 44.0645, Z -4.6667, A 0.000, B 0.000, C 0.000 }
gfCNCPoint3[20410] = {X 589.3408, Y 43.1363, Z -4.6667, A 0.000, B 0.000, C 0.000 }
gfCNCPoint3[20411] = {X 589.6404, Y 42.2516, Z -4.6667, A 0.000, B 0.000, C 0.000 }
gfCNCPoint3[20412] = {X 590.1216, Y 41.4510, Z -4.6667, A 0.000, B 0.000, C 0.000 }
gfCNCPoint3[20413] = {X 590.7622, Y 40.7712, Z -4.6667, A 0.000, B 0.000, C 0.000 }
gfCNCPoint3[20414] = {X 590.7627, Y 33.5311, Z -4.6667, A 0.000, B 0.000, C 0.000 }
gfCNCPoint3[20415] = {X 585.4453, Y 46.6524, Z -4.6667, A 0.000, B 0.000, C 0.000 }
gfCNCPoint3[20416] = {X 585.0755, Y 47.3550, Z -4.6667, A 0.000, B 0.000, C 0.000 }
gfCNCPoint3[20417] = {X 584.5834, Y 47.9780, Z -4.6667, A 0.000, B 0.000, C 0.000 }
gfCNCPoint3[20418] = {X 583.9856, Y 48.5004, Z -4.6667, A 0.000, B 0.000, C 0.000 }
